(* Logix 5000 project; controller Generic 1768-L43 rev 16.2; software revision 15.01 *)

TASK T00_Main (continuous, watchdog 500 ms) : PZ_GenericMachine_AUTO, PZ_GenericMachine_MANUAL, P00_Control, P01_AXIS_00
TASK T02_AXIS_History (periodic, rate 48 ms, priority 10, watchdog 500 ms) : AXIS_EventLog

MODULES
   Local : 1768-L43 (1768Ctrl3Slot 0, Compact 0, rev 16.2)
      SERCOS : 1768-M04SE (1768 1, rev 16.1, MotionAsync RPI 25 ms, MotionEvent RPI 1000 ms, MotionSync RPI 2 ms)
END_MODULES

TYPE UDT_Axis_CMD :
STRUCT
   Enable : BOOL;   // 1=Turn Axis Servo Loop ON
   Disable : BOOL;   // 1=Turn Axis Servo Loop OFF
   Reset : BOOL;   // 1=Clear Axis Faults
   JogFWD : BOOL;   // 1=Jog Forward Direction
   JogREV : BOOL;   // 1=Jog Reverse Direction
   ReferenceREQ : BOOL;   // 1=Set Absolute Reference
END_STRUCT
END_TYPE

TYPE UDT_Axis_Data :
STRUCT
   MoveDir : DINT[8];
   MoveSpd : DINT[8];
   MoveAccel : DINT[8];
   MoveDecel : DINT[8];
   JogDir : DINT[8];
   JogSpd : DINT[8];
   JogAccel : DINT[8];
   JogDecel : DINT[8];
   Direction : DINT[8];
   Offset : REAL[4];
   Dwell : TIMER[16];
   JogTime : TIMER[16];
   InitSEQ : DINT;
   RunSEQ : DINT[4];
   StopSEQ : DINT;
   CamCalcSEQ : DINT;
END_STRUCT
END_TYPE

TYPE UDT_Axis_Status :
STRUCT
   Enabled : BOOL;   // 1=Axis Servo Loop is Active
   OK : BOOL;   // 1=Axis is NOT Faulted
   Auto : BOOL;   // 1=Axis has Attained the Auto Status Means
   Jogging : BOOL;   // 1=Axis is Jogging
   No_Motion : BOOL;   // 1=Axis is Stationary
   Homed : BOOL;   // 1=Axis has been Homed
   Axis_Selected : BOOL;   // 1=Axis to be Active When in Run Mode
   Gear_Active : BOOL;   // 1=Axis is Actively Geared to Another Axis
   Cam_Active : BOOL;   // 1=Axis is Actively Camming
   Move_Active : BOOL;   // 1=Axis is Actively Performing a Move
   Initialized : BOOL;   // 1=Axis has been Initialized
   ConfigComplete : BOOL;   // 1=Axis has been Configured
   ConfigState : DINT;   // Axis Configuration State
END_STRUCT
END_TYPE

TYPE UDT_AxisHistory_CTRL :
STRUCT
   Index : DINT;
   Date_Time : DINT[7];
   Next_Fault : DINT;
   MASR : MOTION_INSTRUCTION;
   Clear_History : BOOL;
   Latch_Bit : BOOL;
   ONS : DINT;
   SourceData : UDT_AxisHistory_DLM;
   Garbage : UDT_AxisHistory_DLM;
   FFL_FFU : CONTROL;
   Update_DLAY : TIMER;
   DLM_LoadDwell : TIMER[2];
END_STRUCT
END_TYPE

TYPE UDT_AxisHistory_DLM :
STRUCT
   SERCOS_NODE : DINT;
   Year : DINT;
   Month : DINT;
   Day : DINT;
   Hour : DINT;
   Minute : DINT;
   Second : DINT;
   GroupStatus : DINT;
   InhibStatus : DINT;
   GroupSynced : DINT;
   GroupFault : DINT;
   GroupOverlapFault : DINT;
   CSTLossFault : DINT;
   GroupTaskLoadingFault : DINT;
   GroupAxisFault : DINT;
   PhysicalAxisFault_Group : DINT;
   ModuleFault_Group : DINT;
   ConfigFault_Group : DINT;
   AxisFault : DINT;
   PhysicalAxisFault : DINT;
   ModuleFault : DINT;
   ConfigFault : DINT;
   ModuleFaults : DINT;
   ControlSyncFault : DINT;
   ModuleSyncFault : DINT;
   TimerEventFault : DINT;
   ModuleHardwareFault : DINT;
   SERCOSRingFault : DINT;
   AttributeErrorCode : DINT;
   AttributeErrorID : DINT;
   InhibitStatus : DINT;
   BusReadyStatus : DINT;
   DriveFault : DINT;
   PosSoftOvertravelFault : DINT;
   NegSoftOvertravelFault : DINT;
   PosHardOvertravelFault : DINT;
   NegHardOvertravelFault : DINT;
   MotFeedbackFault : DINT;
   MotFeedbackNoiseFault : DINT;
   AuxFeedbackFault : DINT;
   AuxFeedbackNoiseFault : DINT;
   DriveEnableInputFault : DINT;
   CommonBusFault : DINT;
   PreChargeOverloadFault : DINT;
   GroundShortFault : DINT;
   DriveHardFault : DINT;
   OverSpeedFault : DINT;
   OverloadFault : DINT;
   DriveOvertempFault : DINT;
   MotorOvertempFault : DINT;
   DriveCoolingFault : DINT;
   DriveControlVoltageFault : DINT;
   FeedbackFault : DINT;
   CommutationFault : DINT;
   DriveOvercurrentFault : DINT;
   DriveOvervoltageFault : DINT;
   DriveUndervoltageFault : DINT;
   PowerPhaseLossFault : DINT;
   PositionErrorFault : DINT;
   SERCOSFault : DINT;
   SERCOSErrorCode : DINT;
END_STRUCT
END_TYPE

TYPE UDT_Machine_COND :
STRUCT
   Networks_Ok : BOOL;
   ESTOP_OK : BOOL;
   GUARDS_OK : BOOL;
   LIGHT_CURTAIN_OK : BOOL;
   ALL_SAFETYs_OK : BOOL;
   All_Axes_Ok : BOOL;
   All_Axes_On : BOOL;
   All_Axes_Off : BOOL;
   All_Axes_Homed : BOOL;
   Home_Permissive : BOOL;
   Any_Line_Start_Pressed : BOOL;
   Any_Line_Stop_Pressed : BOOL;
   Any_Home_Request : BOOL;
   Any_Hold_Pressed : BOOL;
   Auto_Run_State_Active : BOOL;
   All_Axes_Running : BOOL;
   All_Axes_Initialized : BOOL;
   Init_Permissive : BOOL;
   All_Axes_Configured : BOOL;
   All_Axes_Bus_Ok : BOOL;
END_STRUCT
END_TYPE

TYPE UDT_Motion_Instructions :
STRUCT
   MASR : MOTION_INSTRUCTION;
   MAFR : MOTION_INSTRUCTION;
   MSO : MOTION_INSTRUCTION;
   MSF : MOTION_INSTRUCTION;
   MAH : MOTION_INSTRUCTION;
   MRP : MOTION_INSTRUCTION;
   MAJ : MOTION_INSTRUCTION[16];
   MAM : MOTION_INSTRUCTION[16];
   MAG : MOTION_INSTRUCTION[5];
   MCCP : MOTION_INSTRUCTION[5];
   MAPC : MOTION_INSTRUCTION[5];
   MAS : MOTION_INSTRUCTION[16];
   MCD : MOTION_INSTRUCTION;
   MAR : MOTION_INSTRUCTION;
   MDR : MOTION_INSTRUCTION;
END_STRUCT
END_TYPE

TYPE UDT_PhaseTimeout :
STRUCT
   Aborting : TIMER;
   Holding : TIMER;
   Resetting : TIMER;
   Restarting : TIMER;
   Running : TIMER;
   Stopping : TIMER;
END_STRUCT
END_TYPE

VAR_GLOBAL   (* controller tags *)
   AXIS_00 : AXIS_VIRTUAL;
   Axis_00_CMD : UDT_Axis_CMD := (Enable := 1);
   Axis_00_Data : UDT_Axis_Data := (MoveSpd[0] := 10, MoveSpd[1] := 20, MoveSpd[2] := 80, MoveSpd[3] := 90, MoveSpd[4] := 90, MoveAccel[0] := 50, MoveAccel[1] := 50, MoveAccel[2] := 30, MoveAccel[3] := 30, MoveAccel[4] := 40, MoveDecel[0] := 50, JogSpd[0] := 10, JogSpd[1] := 30, JogAccel[0] := 50, JogAccel[1] := 50, JogDecel[0] := 50, JogDecel[1] := 50, Direction[1] := 1, Direction[3] := 1, Dwell[0].PRE := 1500, Dwell[0].ACC := 1501, Dwell[0].EN := 1, Dwell[0].DN := 1, Dwell[1].PRE := 1500, Dwell[2].PRE := 1500, Dwell[2].ACC := 1502, Dwell[2].EN := 1, Dwell[2].DN := 1, Dwell[3].PRE := 1500, Dwell[3].ACC := 1501, Dwell[3].EN := 1, Dwell[3].DN := 1, Dwell[4].PRE := 1500, Dwell[4].ACC := 1500, Dwell[4].EN := 1, Dwell[4].DN := 1, JogTime[0].PRE := 5000, JogTime[1].PRE := 5000, JogTime[2].PRE := 5000, JogTime[3].PRE := 5000, JogTime[4].PRE := 5000);
   Axis_00_MI : UDT_Motion_Instructions := (MASR.FLAGS := 33554432, MAFR.FLAGS := 33554432, MSO.FLAGS := 536870912, MSO.DN := 1, MSO.STATE := 1, MSF.FLAGS := 536870912, MSF.DN := 1, MSF.STATUS := 2, MSF.STATE := 1, MAH.FLAGS := 33554432, MRP.FLAGS := 570425344, MRP.DN := 1, MAJ[0].FLAGS := 570425344, MAJ[0].DN := 1, MAJ[1].FLAGS := 33554432, MAJ[2].FLAGS := 33554432, MAJ[3].FLAGS := 570425344, MAJ[3].DN := 1, MAJ[4].FLAGS := 536870912, MAJ[4].DN := 1, MAM[0].FLAGS := 33554432, MAPC[0].FLAGS := 570425344, MAPC[0].DN := 1, MAS[0].FLAGS := 704643072, MAS[0].DN := 1, MAS[0].PC := 1, MAS[1].FLAGS := 33554432, MAS[2].FLAGS := 704643072, MAS[2].DN := 1, MAS[2].PC := 1, MAS[3].FLAGS := 704643072, MAS[3].DN := 1, MAS[3].PC := 1, MAS[4].FLAGS := 671088640, MAS[4].DN := 1, MAS[4].PC := 1);
   Axis_00_Status : UDT_Axis_Status := (Enabled := 1, OK := 1, Axis_Selected := 1, ConfigComplete := 1, ConfigState := 128);
   AXIS_01 : AXIS_SERVO_DRIVE;
   Axis_01_CMD : UDT_Axis_CMD;
   Axis_01_Data : UDT_Axis_Data := (MoveSpd[0] := 10, MoveSpd[1] := 20, MoveSpd[2] := 80, MoveSpd[3] := 90, MoveSpd[4] := 90, MoveAccel[0] := 50, MoveAccel[1] := 50, MoveAccel[2] := 30, MoveAccel[3] := 30, MoveAccel[4] := 40, MoveDecel[0] := 10, JogSpd[0] := 10, JogSpd[1] := 30, JogAccel[0] := 50, JogAccel[1] := 50, JogDecel[0] := 10, JogDecel[1] := 10, Direction[3] := 1, Dwell[0].PRE := 1500, Dwell[0].ACC := 1501, Dwell[0].EN := 1, Dwell[0].DN := 1, Dwell[1].PRE := 1500, Dwell[2].PRE := 1500, Dwell[2].ACC := 1502, Dwell[2].EN := 1, Dwell[2].DN := 1, Dwell[3].PRE := 1500, Dwell[3].ACC := 1501, Dwell[3].EN := 1, Dwell[3].DN := 1, Dwell[4].PRE := 1500, Dwell[4].ACC := 1500, Dwell[4].EN := 1, Dwell[4].DN := 1, JogTime[0].PRE := 5000, JogTime[1].PRE := 5000, JogTime[2].PRE := 5000, JogTime[3].PRE := 5000, JogTime[4].PRE := 5000);
   Axis_01_MI : UDT_Motion_Instructions := (MASR.FLAGS := 33554432, MAFR.FLAGS := 536870912, MAFR.DN := 1, MSO.FLAGS := 536870912, MSO.DN := 1, MSO.STATE := 1, MSF.FLAGS := 536870912, MSF.DN := 1, MSF.STATUS := 2, MSF.STATE := 1, MAH.FLAGS := 33554432, MAJ[0].FLAGS := 570425344, MAJ[0].DN := 1, MAJ[1].FLAGS := 33554432, MAJ[2].FLAGS := 33554432, MAJ[3].FLAGS := 570425344, MAJ[3].DN := 1, MAJ[4].FLAGS := 536870912, MAJ[4].DN := 1, MAM[0].FLAGS := 704643072, MAM[0].DN := 1, MAM[0].PC := 1, MAPC[0].FLAGS := 570425344, MAPC[0].DN := 1, MAS[0].FLAGS := 33554432, MAS[1].FLAGS := 33554432, MAS[2].FLAGS := 704643072, MAS[2].DN := 1, MAS[2].PC := 1, MAS[3].FLAGS := 704643072, MAS[3].DN := 1, MAS[3].PC := 1, MAS[4].FLAGS := 671088640, MAS[4].DN := 1, MAS[4].PC := 1);
   Axis_01_Status : UDT_Axis_Status := (OK := 1, Axis_Selected := 1, ConfigComplete := 1, ConfigState := 128);
   AXIS_02 : AXIS_SERVO_DRIVE;
   Axis_02_CMD : UDT_Axis_CMD;
   Axis_02_Data : UDT_Axis_Data := (MoveSpd[0] := 10, MoveSpd[1] := 20, MoveSpd[2] := 80, MoveSpd[3] := 90, MoveSpd[4] := 90, MoveAccel[0] := 50, MoveAccel[1] := 50, MoveAccel[2] := 30, MoveAccel[3] := 30, MoveAccel[4] := 40, MoveDecel[0] := 10, JogSpd[0] := 10, JogSpd[1] := 30, JogAccel[0] := 50, JogAccel[1] := 50, JogDecel[0] := 10, JogDecel[1] := 10, Direction[3] := 1, Dwell[0].PRE := 1500, Dwell[1].PRE := 1500, Dwell[2].PRE := 1500, Dwell[2].ACC := 1501, Dwell[2].EN := 1, Dwell[2].DN := 1, Dwell[3].PRE := 1500, Dwell[3].ACC := 1501, Dwell[3].EN := 1, Dwell[3].DN := 1, Dwell[4].PRE := 1500, Dwell[4].ACC := 1502, Dwell[4].EN := 1, Dwell[4].DN := 1, JogTime[0].PRE := 5000, JogTime[0].ACC := 4648, JogTime[0].EN := 1, JogTime[0].TT := 1, JogTime[1].PRE := 5000, JogTime[2].PRE := 5000, JogTime[3].PRE := 5000, JogTime[4].PRE := 5000);
   Axis_02_MI : UDT_Motion_Instructions := (MASR.FLAGS := 33554432, MAFR.FLAGS := 536870912, MAFR.DN := 1, MSO.FLAGS := 536870912, MSO.DN := 1, MSO.STATE := 1, MSF.FLAGS := 536870912, MSF.DN := 1, MSF.STATUS := 2, MSF.STATE := 1, MAH.FLAGS := 33554432, MAJ[0].FLAGS := 570425344, MAJ[0].DN := 1, MAJ[1].FLAGS := 33554432, MAJ[2].FLAGS := 33554432, MAJ[3].FLAGS := 570425344, MAJ[3].DN := 1, MAJ[4].FLAGS := 536870912, MAJ[4].DN := 1, MAM[0].FLAGS := 704643072, MAM[0].DN := 1, MAM[0].PC := 1, MAS[0].FLAGS := 33554432, MAS[1].FLAGS := 33554432, MAS[2].FLAGS := 704643072, MAS[2].DN := 1, MAS[2].PC := 1, MAS[3].FLAGS := 704643072, MAS[3].DN := 1, MAS[3].PC := 1, MAS[4].FLAGS := 671088640, MAS[4].DN := 1, MAS[4].PC := 1);
   Axis_02_Status : UDT_Axis_Status := (Axis_Selected := 1, ConfigComplete := 1, ConfigState := 128);
   AXIS_03 : AXIS_SERVO_DRIVE;
   Axis_03_CMD : UDT_Axis_CMD;
   Axis_03_Data : UDT_Axis_Data := (MoveSpd[0] := 10, MoveSpd[1] := 20, MoveSpd[2] := 80, MoveSpd[3] := 90, MoveSpd[4] := 90, MoveAccel[0] := 50, MoveAccel[1] := 50, MoveAccel[2] := 30, MoveAccel[3] := 30, MoveAccel[4] := 40, MoveDecel[0] := 10, JogSpd[0] := 10, JogSpd[1] := 30, JogAccel[0] := 50, JogAccel[1] := 50, JogDecel[0] := 10, JogDecel[1] := 10, Direction[3] := 1, Dwell[0].PRE := 1500, Dwell[1].PRE := 1500, Dwell[2].PRE := 1500, Dwell[2].ACC := 1501, Dwell[2].EN := 1, Dwell[2].DN := 1, Dwell[3].PRE := 1500, Dwell[3].ACC := 1501, Dwell[3].EN := 1, Dwell[3].DN := 1, Dwell[4].PRE := 1500, Dwell[4].ACC := 1502, Dwell[4].EN := 1, Dwell[4].DN := 1, JogTime[0].PRE := 5000, JogTime[0].ACC := 4648, JogTime[0].EN := 1, JogTime[0].TT := 1, JogTime[1].PRE := 5000, JogTime[2].PRE := 5000, JogTime[3].PRE := 5000, JogTime[4].PRE := 5000);
   Axis_03_MI : UDT_Motion_Instructions := (MASR.FLAGS := 33554432, MAFR.FLAGS := 536870912, MAFR.DN := 1, MSO.FLAGS := 536870912, MSO.DN := 1, MSO.STATE := 1, MSF.FLAGS := 536870912, MSF.DN := 1, MSF.STATUS := 2, MSF.STATE := 1, MAH.FLAGS := 33554432, MAJ[0].FLAGS := 570425344, MAJ[0].DN := 1, MAJ[1].FLAGS := 33554432, MAJ[2].FLAGS := 33554432, MAJ[3].FLAGS := 570425344, MAJ[3].DN := 1, MAJ[4].FLAGS := 536870912, MAJ[4].DN := 1, MAM[0].FLAGS := 704643072, MAM[0].DN := 1, MAM[0].PC := 1, MAS[0].FLAGS := 33554432, MAS[1].FLAGS := 33554432, MAS[2].FLAGS := 704643072, MAS[2].DN := 1, MAS[2].PC := 1, MAS[3].FLAGS := 704643072, MAS[3].DN := 1, MAS[3].PC := 1, MAS[4].FLAGS := 671088640, MAS[4].DN := 1, MAS[4].PC := 1);
   Axis_03_Status : UDT_Axis_Status := (Axis_Selected := 1, ConfigComplete := 1, ConfigState := 128);
   AXIS_04 : AXIS_SERVO_DRIVE;
   Axis_04_CMD : UDT_Axis_CMD;
   Axis_04_Data : UDT_Axis_Data := (MoveSpd[0] := 10, MoveSpd[1] := 20, MoveSpd[2] := 80, MoveSpd[3] := 90, MoveSpd[4] := 90, MoveAccel[0] := 50, MoveAccel[1] := 50, MoveAccel[2] := 30, MoveAccel[3] := 30, MoveAccel[4] := 40, MoveDecel[0] := 10, JogSpd[0] := 10, JogSpd[1] := 30, JogAccel[0] := 50, JogAccel[1] := 50, JogDecel[0] := 10, JogDecel[1] := 10, Direction[3] := 1, Dwell[0].PRE := 1500, Dwell[1].PRE := 1500, Dwell[2].PRE := 1500, Dwell[2].ACC := 1501, Dwell[2].EN := 1, Dwell[2].DN := 1, Dwell[3].PRE := 1500, Dwell[3].ACC := 1501, Dwell[3].EN := 1, Dwell[3].DN := 1, Dwell[4].PRE := 1500, Dwell[4].ACC := 1502, Dwell[4].EN := 1, Dwell[4].DN := 1, JogTime[0].PRE := 5000, JogTime[0].ACC := 4648, JogTime[0].EN := 1, JogTime[0].TT := 1, JogTime[1].PRE := 5000, JogTime[2].PRE := 5000, JogTime[3].PRE := 5000, JogTime[4].PRE := 5000);
   Axis_04_MI : UDT_Motion_Instructions := (MASR.FLAGS := 33554432, MAFR.FLAGS := 536870912, MAFR.DN := 1, MSO.FLAGS := 536870912, MSO.DN := 1, MSO.STATE := 1, MSF.FLAGS := 536870912, MSF.DN := 1, MSF.STATUS := 2, MSF.STATE := 1, MAH.FLAGS := 33554432, MAJ[0].FLAGS := 570425344, MAJ[0].DN := 1, MAJ[1].FLAGS := 33554432, MAJ[2].FLAGS := 33554432, MAJ[3].FLAGS := 570425344, MAJ[3].DN := 1, MAJ[4].FLAGS := 536870912, MAJ[4].DN := 1, MAM[0].FLAGS := 704643072, MAM[0].DN := 1, MAM[0].PC := 1, MAS[0].FLAGS := 33554432, MAS[1].FLAGS := 33554432, MAS[2].FLAGS := 704643072, MAS[2].DN := 1, MAS[2].PC := 1, MAS[3].FLAGS := 704643072, MAS[3].DN := 1, MAS[3].PC := 1, MAS[4].FLAGS := 671088640, MAS[4].DN := 1, MAS[4].PC := 1);
   Axis_04_Status : UDT_Axis_Status := (Axis_Selected := 1, ConfigComplete := 1, ConfigState := 128);
   AXIS_Servo_Generic : AXIS_SERVO_DRIVE;
   C_pi : REAL := 3.1415927;
   ClearFaultDelay : TIMER := (PRE := 250);
   GenericMachine_COND : UDT_Machine_COND := (Networks_Ok := 1, ESTOP_OK := 1, GUARDS_OK := 1, LIGHT_CURTAIN_OK := 1, ALL_SAFETYs_OK := 1, All_Axes_Off := 1, Init_Permissive := 1, All_Axes_Configured := 1, All_Axes_Bus_Ok := 1);
   GUI_Axis_01_JogFwdREQ : BOOL;
   GUI_Axis_01_JogRevREQ : BOOL;
   GUI_Axis_01_ReferenceREQ : BOOL;
   GUI_Axis_02_JogFwdREQ : BOOL;
   GUI_Axis_02_JogRevREQ : BOOL;
   GUI_Axis_02_ReferenceREQ : BOOL;
   GUI_Axis_03_JogFwdREQ : BOOL;
   GUI_Axis_03_JogRevREQ : BOOL;
   GUI_Axis_03_ReferenceREQ : BOOL;
   GUI_Axis_04_JogFwdREQ : BOOL;
   GUI_Axis_04_JogRevREQ : BOOL;
   GUI_Axis_04_ReferenceREQ : BOOL;
   GUI_HoldRequest : BOOL;
   GUI_JogFwdRequest : BOOL;
   GUI_JogRevRequest : BOOL;
   GUI_ManualABSrefStatDISP : DINT := 1;
   GUI_ManualAxisSelect : DINT;
   GUI_ManualControlRequest : BOOL;
   GUI_ManualPositionDISP : REAL := 0.334165;
   GUI_ManualSASDISP : DINT;
   GUI_ManualVelocityDISP : REAL;
   GUI_ReferenceREQ : BOOL;
   GUI_RunSPD_NI : DINT := 5;
   GUI_ServoReReferenceRequest : BOOL;
   GUI_StartRequest : BOOL;
   GUI_StopRequest : BOOL;
   ManualControl : BOOL;
   MASK : DINT := -1;
   MotionGroup : MOTION_GROUP;
   PhaseTimout : UDT_PhaseTimeout := (Aborting.PRE := 5000, Holding.PRE := 5000, Resetting.PRE := 5000, Restarting.PRE := 5000, Stopping.PRE := 5000);
   PowerUP_TMR : TIMER := (PRE := 10000, ACC := 10000);
   PZ_GenericMachine_AUTO : PHASE := (State := 1024, Aborted := 1);
   PZ_GenericMachine_MANUAL : PHASE := (State := 512, Stopped := 1);
END_VAR

PROGRAM AXIS_EventLog   (* main routine R00_Dispatch *)
VAR
   EL_CTRL_1 : UDT_AxisHistory_CTRL := (Date_Time[0] := 1998, Date_Time[1] := 1, Date_Time[2] := 4, Date_Time[3] := 14, Date_Time[4] := 48, Date_Time[5] := 48, Date_Time[6] := 956843, SourceData.SERCOS_NODE := 1, SourceData.Year := 1998, SourceData.Month := 1, SourceData.Day := 4, SourceData.Hour := 14, SourceData.Minute := 48, SourceData.Second := 48, SourceData.GroupStatus := 16#0000_0006, SourceData.GroupSynced := 1, SourceData.GroupAxisFault := 16#0000_0001, SourceData.PhysicalAxisFault_Group := 1, SourceData.AxisFault := 16#0000_0001, SourceData.PhysicalAxisFault := 1, SourceData.DriveFault := 16#0800_0000, SourceData.PositionErrorFault := 1, FFL_FFU.LEN := 51, FFL_FFU.POS := 50, Update_DLAY.PRE := 24, DLM_LoadDwell[0].PRE := 1000, DLM_LoadDwell[1].PRE := 1000);
   EL_CTRL_2 : UDT_AxisHistory_CTRL := (Date_Time[0] := 1998, Date_Time[1] := 1, Date_Time[2] := 4, Date_Time[3] := 14, Date_Time[4] := 54, Date_Time[5] := 19, Date_Time[6] := 52840, Next_Fault := 3, ONS := 1, SourceData.SERCOS_NODE := 2, SourceData.Year := 1998, SourceData.Month := 1, SourceData.Day := 4, SourceData.Hour := 14, SourceData.Minute := 54, SourceData.Second := 19, SourceData.GroupStatus := 16#0000_0006, SourceData.GroupSynced := 1, SourceData.GroupAxisFault := 16#0000_0001, SourceData.PhysicalAxisFault_Group := 1, SourceData.AxisFault := 16#0000_0001, SourceData.PhysicalAxisFault := 1, SourceData.DriveFault := 16#0800_0000, SourceData.PositionErrorFault := 1, FFL_FFU.LEN := 51, FFL_FFU.POS := 50, Update_DLAY.PRE := 24, Update_DLAY.ACC := 48, Update_DLAY.EN := 1, Update_DLAY.DN := 1, DLM_LoadDwell[0].PRE := 1000, DLM_LoadDwell[1].PRE := 1000);
   EL_CTRL_3 : UDT_AxisHistory_CTRL := (Date_Time[0] := 1998, Date_Time[1] := 1, Date_Time[2] := 1, Date_Time[3] := 15, Date_Time[4] := 41, Date_Time[5] := 17, Date_Time[6] := 485526, FFL_FFU.LEN := 51, FFL_FFU.POS := 50, FFL_FFU.EN := 1, FFL_FFU.EU := 1, Update_DLAY.PRE := 24, DLM_LoadDwell[0].PRE := 1000, DLM_LoadDwell[1].PRE := 1000);
   EL_CTRL_4 : UDT_AxisHistory_CTRL := (Date_Time[0] := 1998, Date_Time[1] := 1, Date_Time[2] := 1, Date_Time[3] := 15, Date_Time[4] := 41, Date_Time[5] := 17, Date_Time[6] := 437605, FFL_FFU.LEN := 51, FFL_FFU.POS := 50, FFL_FFU.EN := 1, FFL_FFU.EU := 1, Update_DLAY.PRE := 24, DLM_LoadDwell[0].PRE := 1000, DLM_LoadDwell[1].PRE := 1000);
   EL_CTRL_5 : UDT_AxisHistory_CTRL := (Date_Time[0] := 1998, Date_Time[1] := 1, Date_Time[2] := 1, Date_Time[3] := 15, Date_Time[4] := 41, Date_Time[5] := 17, Date_Time[6] := 438340, FFL_FFU.LEN := 51, FFL_FFU.POS := 50, FFL_FFU.EN := 1, FFL_FFU.EU := 1, Update_DLAY.PRE := 24, DLM_LoadDwell[0].PRE := 1000, DLM_LoadDwell[1].PRE := 1000);
   EL_CTRL_6 : UDT_AxisHistory_CTRL := (FFL_FFU.LEN := 51, FFL_FFU.POS := 50, FFL_FFU.EN := 1, FFL_FFU.EU := 1, Update_DLAY.PRE := 24, DLM_LoadDwell[0].PRE := 1000, DLM_LoadDwell[1].PRE := 1000);
   EL_CTRL_7 : UDT_AxisHistory_CTRL := (Date_Time[0] := 2006, Date_Time[1] := 2, Date_Time[2] := 9, Date_Time[3] := 17, Date_Time[4] := 41, Date_Time[5] := 26, Date_Time[6] := 391260, SourceData.SERCOS_NODE := 7, SourceData.Year := 2006, SourceData.Month := 2, SourceData.Day := 9, SourceData.Hour := 17, SourceData.Minute := 41, SourceData.Second := 26, SourceData.GroupStatus := 16#0000_0006, SourceData.GroupSynced := 1, SourceData.GroupAxisFault := 16#0000_0001, SourceData.PhysicalAxisFault_Group := 1, SourceData.AxisFault := 16#0000_0001, SourceData.PhysicalAxisFault := 1, SourceData.DriveFault := 16#0800_0000, SourceData.PositionErrorFault := 1, FFL_FFU.LEN := 51, FFL_FFU.POS := 50, FFL_FFU.EN := 1, FFL_FFU.EU := 1, Update_DLAY.PRE := 24, DLM_LoadDwell[0].PRE := 1000, DLM_LoadDwell[1].PRE := 1000);
   EL_CTRL_8 : UDT_AxisHistory_CTRL := (Date_Time[0] := 2006, Date_Time[1] := 2, Date_Time[2] := 9, Date_Time[3] := 17, Date_Time[4] := 43, Date_Time[5] := 28, Date_Time[6] := 567606, SourceData.SERCOS_NODE := 8, SourceData.Year := 2006, SourceData.Month := 2, SourceData.Day := 9, SourceData.Hour := 17, SourceData.Minute := 43, SourceData.Second := 28, SourceData.GroupStatus := 16#0000_0006, SourceData.GroupSynced := 1, SourceData.GroupAxisFault := 16#0000_0001, SourceData.PhysicalAxisFault_Group := 1, SourceData.AxisFault := 16#0000_0001, SourceData.PhysicalAxisFault := 1, SourceData.DriveFault := 16#0800_0000, SourceData.PositionErrorFault := 1, FFL_FFU.LEN := 51, FFL_FFU.POS := 50, FFL_FFU.EN := 1, FFL_FFU.EU := 1, Update_DLAY.PRE := 24, DLM_LoadDwell[0].PRE := 1000, DLM_LoadDwell[1].PRE := 1000);
   EL_SaveSEQ : DINT;
   EventINDEX : DINT;
   EventLog_N1 : UDT_AxisHistory_DLM[51];
   EventLog_N2 : UDT_AxisHistory_DLM[51];
   EventLog_N3 : UDT_AxisHistory_DLM[51];
   EventLog_N4 : UDT_AxisHistory_DLM[51];
   EventLog_N5 : UDT_AxisHistory_DLM[51];
   EventLog_N6 : UDT_AxisHistory_DLM[51];
   EventLog_N7 : UDT_AxisHistory_DLM[51];
   EventLog_N8 : UDT_AxisHistory_DLM[51];
   GUI_DataDisplay : UDT_AxisHistory_DLM;
   GUI_DataLogModel : UDT_AxisHistory_DLM := (SERCOS_NODE := -1, Year := -1, Month := -1, Day := -1, Hour := -1, Minute := -1, Second := -1, GroupStatus := 16#ffff_ffff, InhibStatus := -1, GroupSynced := -1, GroupFault := 16#ffff_ffff, GroupOverlapFault := -1, CSTLossFault := -1, GroupTaskLoadingFault := -1, GroupAxisFault := 16#ffff_ffff, PhysicalAxisFault_Group := -1, ModuleFault_Group := -1, ConfigFault_Group := -1, AxisFault := 16#ffff_ffff, PhysicalAxisFault := -1, ModuleFault := -1, ConfigFault := -1, ModuleFaults := 16#ffff_ffff, ControlSyncFault := -1, ModuleSyncFault := -1, TimerEventFault := -1, ModuleHardwareFault := -1, SERCOSRingFault := -1, AttributeErrorCode := 16#ffff_ffff, AttributeErrorID := 16#ffff_ffff, InhibitStatus := -1, BusReadyStatus := -1, DriveFault := 16#ffff_ffff, PosSoftOvertravelFault := -1, NegSoftOvertravelFault := -1, PosHardOvertravelFault := -1, NegHardOvertravelFault := -1, MotFeedbackFault := -1, MotFeedbackNoiseFault := -1, AuxFeedbackFault := -1, AuxFeedbackNoiseFault := -1, DriveEnableInputFault := -1, CommonBusFault := -1, PreChargeOverloadFault := -1, GroundShortFault := -1, DriveHardFault := -1, OverSpeedFault := -1, OverloadFault := -1, DriveOvertempFault := -1, MotorOvertempFault := -1, DriveCoolingFault := -1, DriveControlVoltageFault := -1, FeedbackFault := -1, CommutationFault := -1, DriveOvercurrentFault := -1, DriveOvervoltageFault := -1, DriveUndervoltageFault := -1, PowerPhaseLossFault := -1, PositionErrorFault := -1, SERCOSFault := -1,
        SERCOSErrorCode := 16#ffff_ffff);
   GUI_EventLogSaving : BOOL;
   GUI_IndexSelect : DINT := 48;
   GUI_NodeSelect : DINT := 8;
   GUI_SaveEventLog : BOOL;
   LogLength : DINT := 51;
   Motion_Group : ALIAS FOR MotionGroup;
   PowerUP_TMR : TIMER := (PRE := 10000, ACC := 10032);
   Servo_Axis_Node_1 : ALIAS FOR AXIS_01;
   Servo_Axis_Node_2 : ALIAS FOR AXIS_02;
   Servo_Axis_Node_3 : ALIAS FOR AXIS_03;
   Servo_Axis_Node_4 : ALIAS FOR AXIS_04;
   Servo_Axis_Node_5 : ALIAS FOR AXIS_Servo_Generic;
   Servo_Axis_Node_6 : ALIAS FOR AXIS_Servo_Generic;
   Servo_Axis_Node_7 : ALIAS FOR AXIS_Servo_Generic;
   Servo_Axis_Node_8 : ALIAS FOR AXIS_Servo_Generic;
END_VAR

ROUTINE R00_Dispatch   (* ladder *)
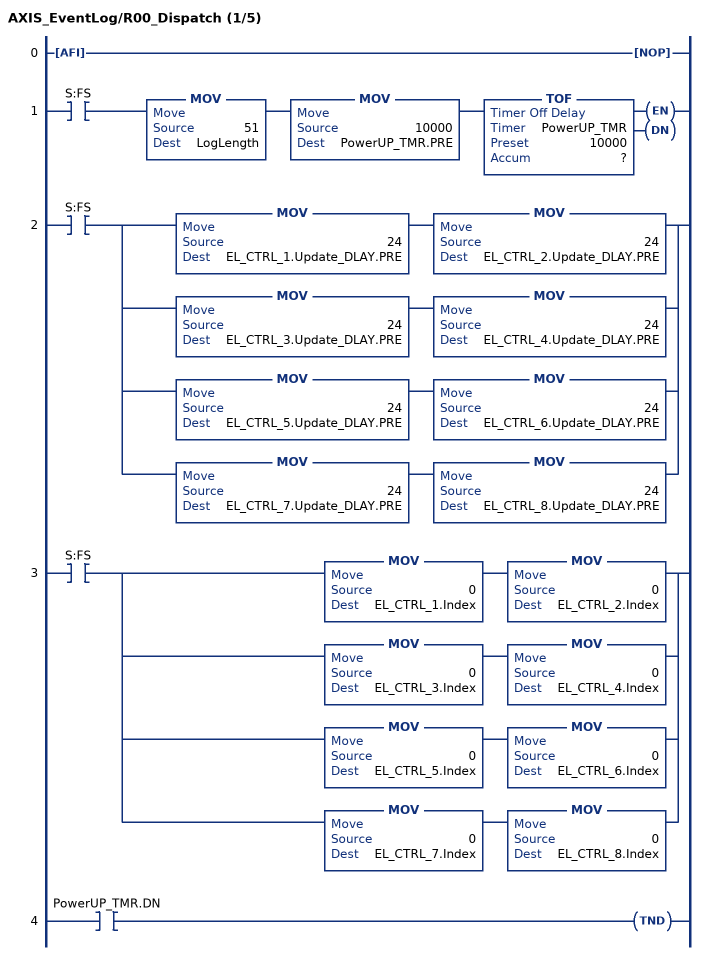
   0: AFI()NOP();
   1: XIC(S:FS)MOV(51,LogLength)MOV(10000,PowerUP_TMR.PRE)TOF(PowerUP_TMR,?,?);
   2: XIC(S:FS)[MOV(24,EL_CTRL_1.Update_DLAY.PRE) MOV(24,EL_CTRL_2.Update_DLAY.PRE) ,MOV(24,EL_CTRL_3.Update_DLAY.PRE) MOV(24,EL_CTRL_4.Update_DLAY.PRE) ,MOV(24,EL_CTRL_5.Update_DLAY.PRE) MOV(24,EL_CTRL_6.Update_DLAY.PRE) ,MOV(24,EL_CTRL_7.Update_DLAY.PRE) MOV(24,EL_CTRL_8.Update_DLAY.PRE) ];
   3: XIC(S:FS)[MOV(0,EL_CTRL_1.Index) MOV(0,EL_CTRL_2.Index) ,MOV(0,EL_CTRL_3.Index) MOV(0,EL_CTRL_4.Index) ,MOV(0,EL_CTRL_5.Index) MOV(0,EL_CTRL_6.Index) ,MOV(0,EL_CTRL_7.Index) MOV(0,EL_CTRL_8.Index) ];
   4: XIC(PowerUP_TMR.DN)TND();
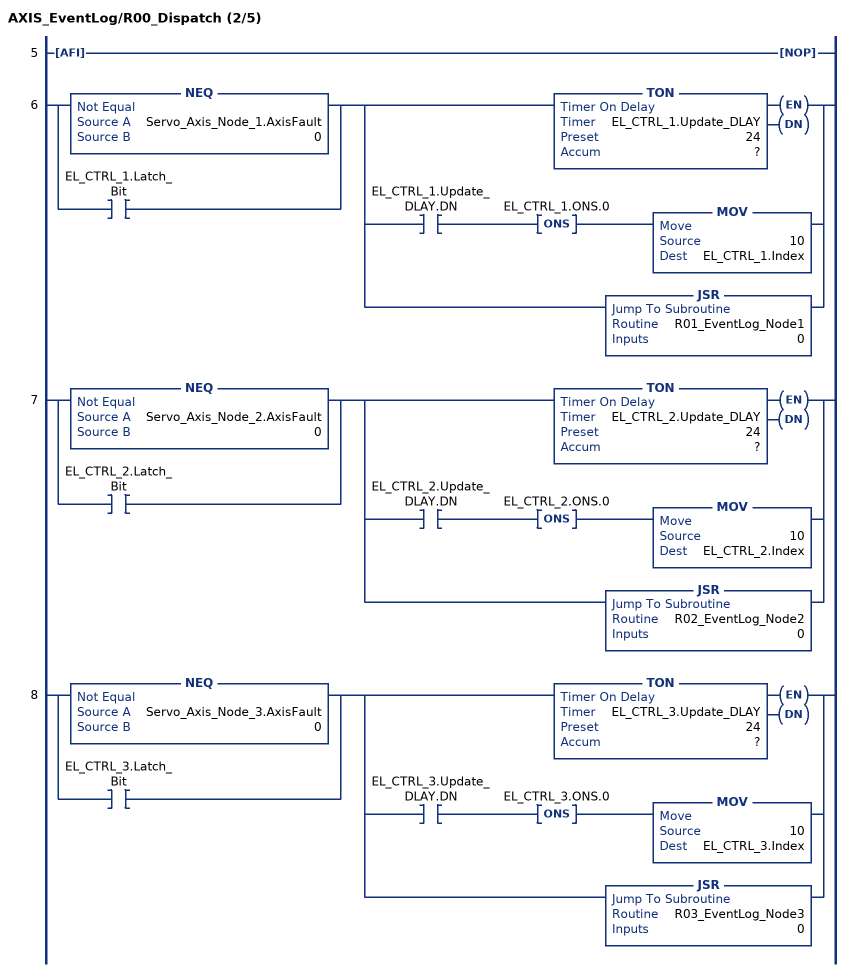
   5: AFI()NOP();
   6: [NEQ(Servo_Axis_Node_1.AxisFault,0) ,XIC(EL_CTRL_1.Latch_Bit) ][TON(EL_CTRL_1.Update_DLAY,?,?) ,XIC(EL_CTRL_1.Update_DLAY.DN) ONS(EL_CTRL_1.ONS.0) MOV(10,EL_CTRL_1.Index) ,JSR(R01_EventLog_Node1,0) ];
   7: [NEQ(Servo_Axis_Node_2.AxisFault,0) ,XIC(EL_CTRL_2.Latch_Bit) ][TON(EL_CTRL_2.Update_DLAY,?,?) ,XIC(EL_CTRL_2.Update_DLAY.DN) ONS(EL_CTRL_2.ONS.0) MOV(10,EL_CTRL_2.Index) ,JSR(R02_EventLog_Node2,0) ];
   8: [NEQ(Servo_Axis_Node_3.AxisFault,0) ,XIC(EL_CTRL_3.Latch_Bit) ][TON(EL_CTRL_3.Update_DLAY,?,?) ,XIC(EL_CTRL_3.Update_DLAY.DN) ONS(EL_CTRL_3.ONS.0) MOV(10,EL_CTRL_3.Index) ,JSR(R03_EventLog_Node3,0) ];
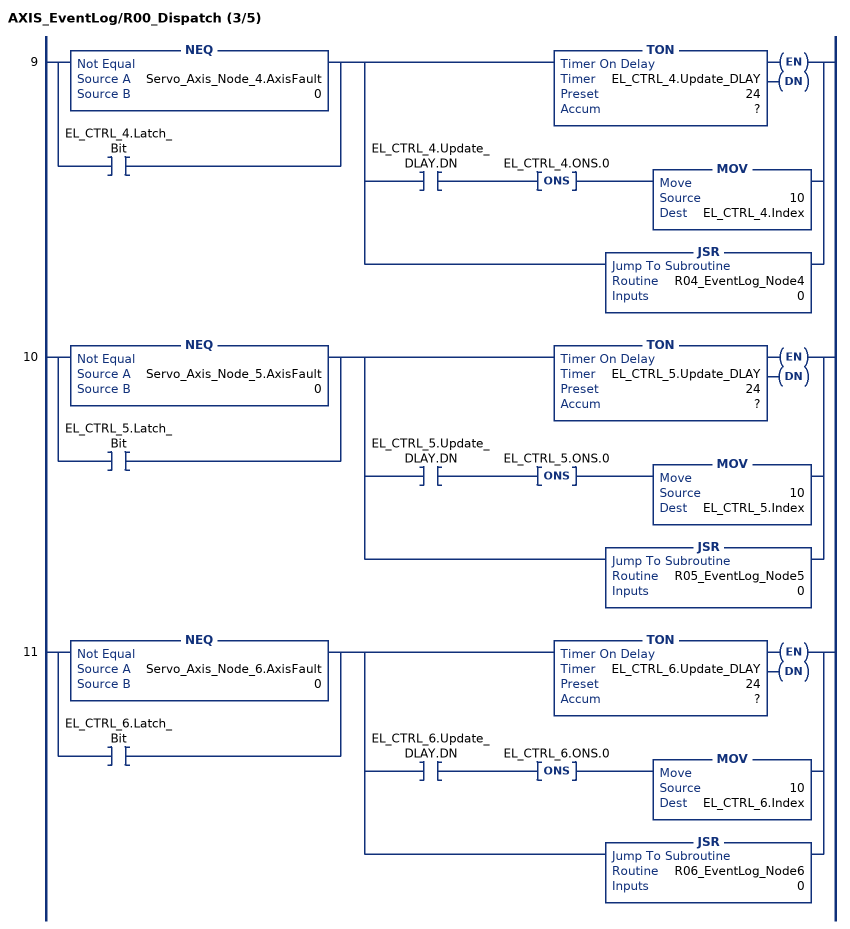
   9: [NEQ(Servo_Axis_Node_4.AxisFault,0) ,XIC(EL_CTRL_4.Latch_Bit) ][TON(EL_CTRL_4.Update_DLAY,?,?) ,XIC(EL_CTRL_4.Update_DLAY.DN) ONS(EL_CTRL_4.ONS.0) MOV(10,EL_CTRL_4.Index) ,JSR(R04_EventLog_Node4,0) ];
   10: [NEQ(Servo_Axis_Node_5.AxisFault,0) ,XIC(EL_CTRL_5.Latch_Bit) ][TON(EL_CTRL_5.Update_DLAY,?,?) ,XIC(EL_CTRL_5.Update_DLAY.DN) ONS(EL_CTRL_5.ONS.0) MOV(10,EL_CTRL_5.Index) ,JSR(R05_EventLog_Node5,0) ];
   11: [NEQ(Servo_Axis_Node_6.AxisFault,0) ,XIC(EL_CTRL_6.Latch_Bit) ][TON(EL_CTRL_6.Update_DLAY,?,?) ,XIC(EL_CTRL_6.Update_DLAY.DN) ONS(EL_CTRL_6.ONS.0) MOV(10,EL_CTRL_6.Index) ,JSR(R06_EventLog_Node6,0) ];
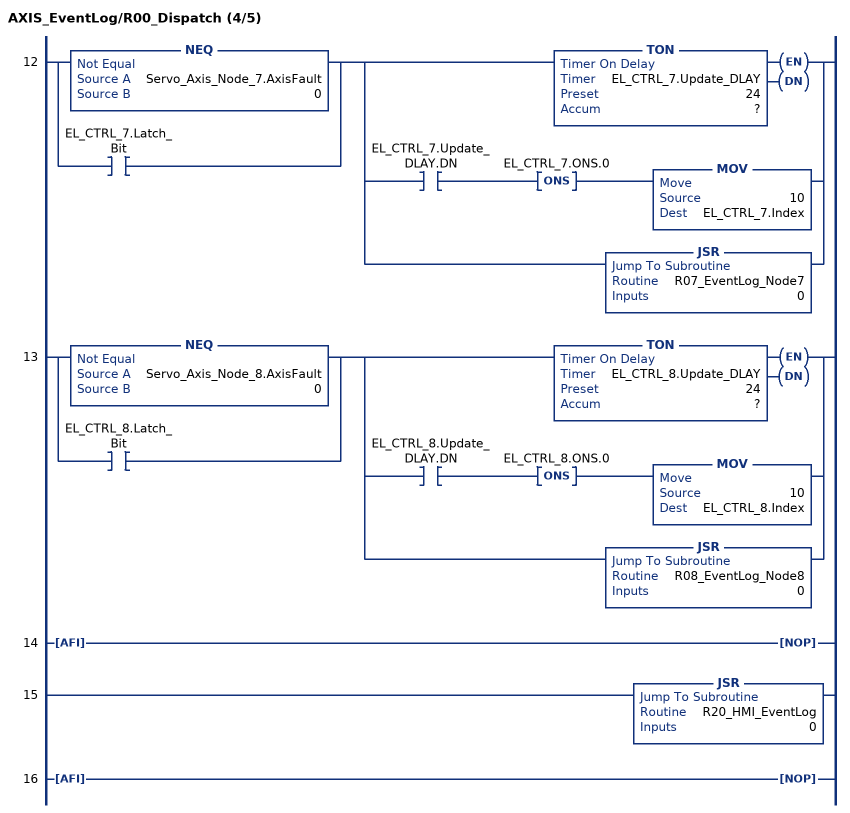
   12: [NEQ(Servo_Axis_Node_7.AxisFault,0) ,XIC(EL_CTRL_7.Latch_Bit) ][TON(EL_CTRL_7.Update_DLAY,?,?) ,XIC(EL_CTRL_7.Update_DLAY.DN) ONS(EL_CTRL_7.ONS.0) MOV(10,EL_CTRL_7.Index) ,JSR(R07_EventLog_Node7,0) ];
   13: [NEQ(Servo_Axis_Node_8.AxisFault,0) ,XIC(EL_CTRL_8.Latch_Bit) ][TON(EL_CTRL_8.Update_DLAY,?,?) ,XIC(EL_CTRL_8.Update_DLAY.DN) ONS(EL_CTRL_8.ONS.0) MOV(10,EL_CTRL_8.Index) ,JSR(R08_EventLog_Node8,0) ];
   14: AFI()NOP();
   15: JSR(R20_HMI_EventLog,0);
   16: AFI()NOP();
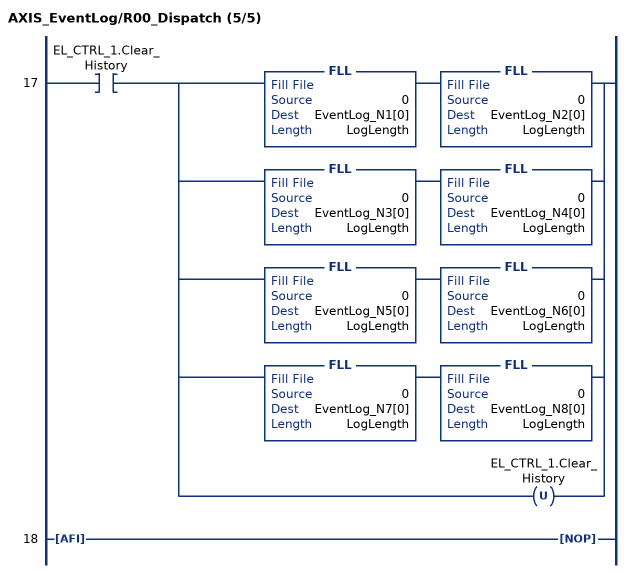
   17: XIC(EL_CTRL_1.Clear_History)[FLL(0,EventLog_N1[0],LogLength) FLL(0,EventLog_N2[0],LogLength) ,FLL(0,EventLog_N3[0],LogLength) FLL(0,EventLog_N4[0],LogLength) ,FLL(0,EventLog_N5[0],LogLength) FLL(0,EventLog_N6[0],LogLength) ,FLL(0,EventLog_N7[0],LogLength) FLL(0,EventLog_N8[0],LogLength) ,OTU(EL_CTRL_1.Clear_History) ];
   18: AFI()NOP();
END_ROUTINE

ROUTINE R01_EventLog_Node1   (* ladder *)
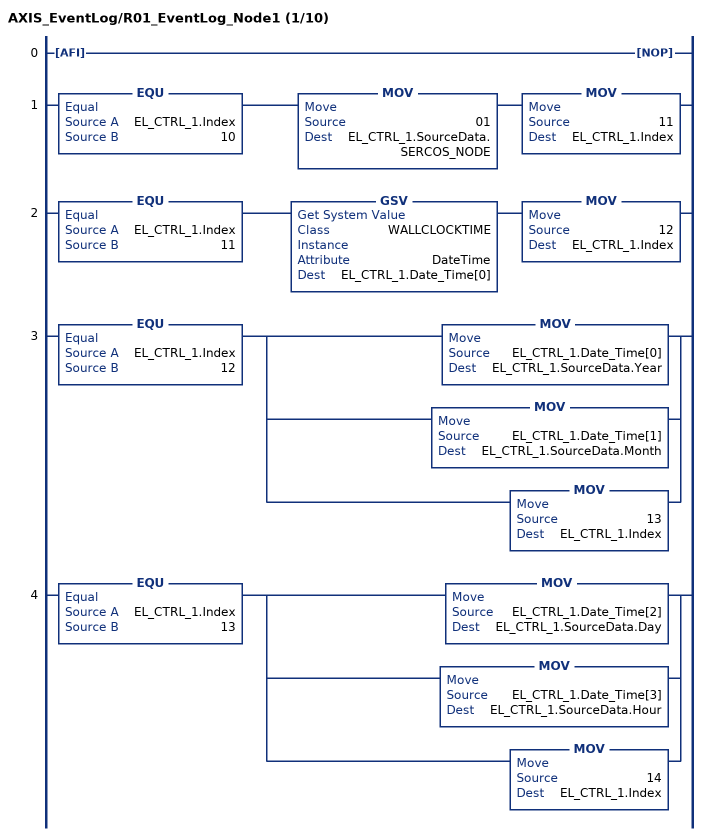
   0: AFI()NOP();
   1: EQU(EL_CTRL_1.Index,10)MOV(01,EL_CTRL_1.SourceData.SERCOS_NODE)MOV(11,EL_CTRL_1.Index);
   2: EQU(EL_CTRL_1.Index,11)GSV(WALLCLOCKTIME,,DateTime,EL_CTRL_1.Date_Time[0])MOV(12,EL_CTRL_1.Index);
   3: EQU(EL_CTRL_1.Index,12)[MOV(EL_CTRL_1.Date_Time[0],EL_CTRL_1.SourceData.Year) ,MOV(EL_CTRL_1.Date_Time[1],EL_CTRL_1.SourceData.Month) ,MOV(13,EL_CTRL_1.Index) ];
   4: EQU(EL_CTRL_1.Index,13)[MOV(EL_CTRL_1.Date_Time[2],EL_CTRL_1.SourceData.Day) ,MOV(EL_CTRL_1.Date_Time[3],EL_CTRL_1.SourceData.Hour) ,MOV(14,EL_CTRL_1.Index) ];
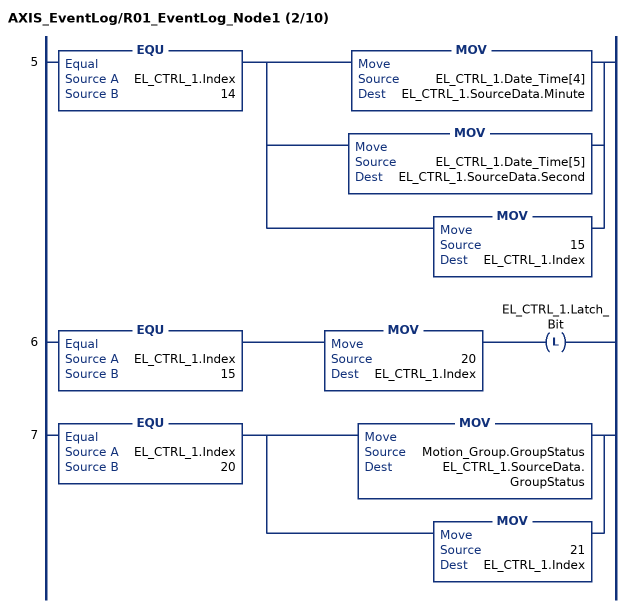
   5: EQU(EL_CTRL_1.Index,14)[MOV(EL_CTRL_1.Date_Time[4],EL_CTRL_1.SourceData.Minute) ,MOV(EL_CTRL_1.Date_Time[5],EL_CTRL_1.SourceData.Second) ,MOV(15,EL_CTRL_1.Index) ];
   6: EQU(EL_CTRL_1.Index,15)MOV(20,EL_CTRL_1.Index)OTL(EL_CTRL_1.Latch_Bit);
   7: EQU(EL_CTRL_1.Index,20)[MOV(Motion_Group.GroupStatus,EL_CTRL_1.SourceData.GroupStatus) ,MOV(21,EL_CTRL_1.Index) ];
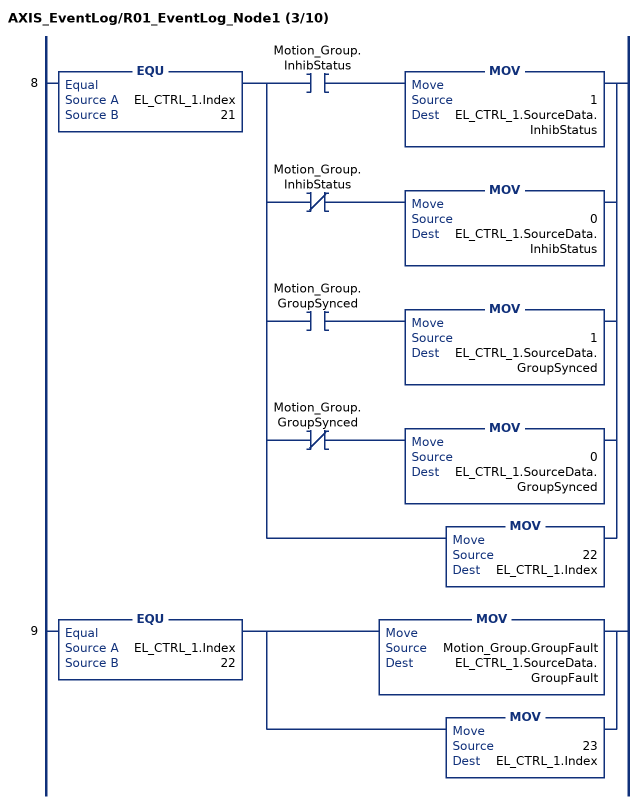
   8: EQU(EL_CTRL_1.Index,21)[XIC(Motion_Group.InhibStatus) MOV(1,EL_CTRL_1.SourceData.InhibStatus) ,XIO(Motion_Group.InhibStatus) MOV(0,EL_CTRL_1.SourceData.InhibStatus) ,XIC(Motion_Group.GroupSynced) MOV(1,EL_CTRL_1.SourceData.GroupSynced) ,XIO(Motion_Group.GroupSynced) MOV(0,EL_CTRL_1.SourceData.GroupSynced) ,MOV(22,EL_CTRL_1.Index) ];
   9: EQU(EL_CTRL_1.Index,22)[MOV(Motion_Group.GroupFault,EL_CTRL_1.SourceData.GroupFault) ,MOV(23,EL_CTRL_1.Index) ];
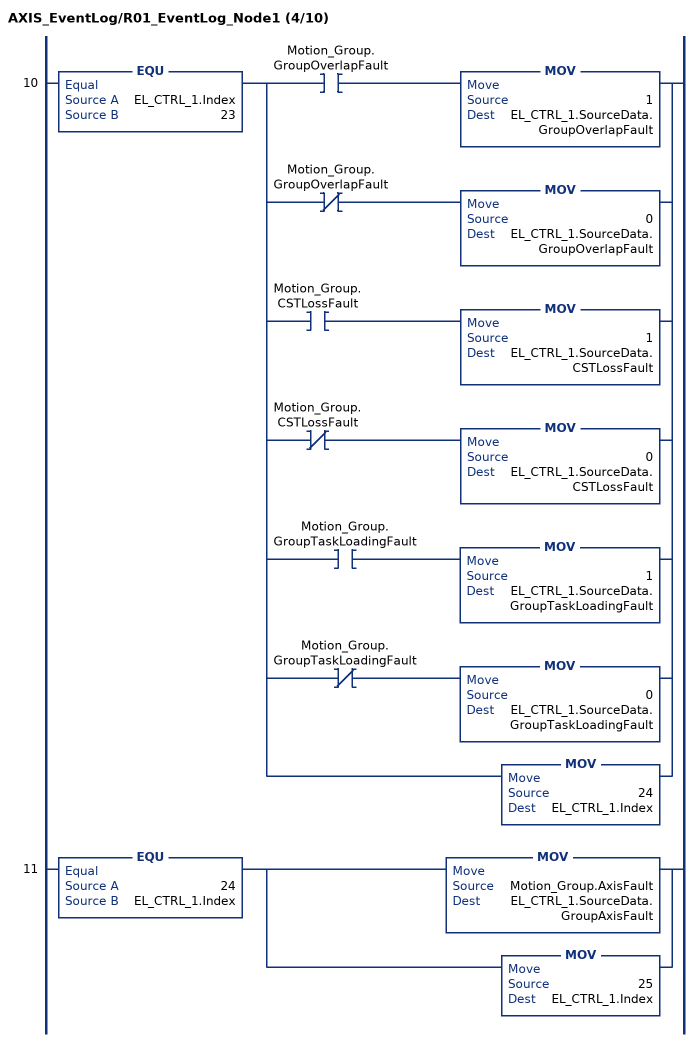
   10: EQU(EL_CTRL_1.Index,23)[XIC(Motion_Group.GroupOverlapFault) MOV(1,EL_CTRL_1.SourceData.GroupOverlapFault) ,XIO(Motion_Group.GroupOverlapFault) MOV(0,EL_CTRL_1.SourceData.GroupOverlapFault) ,XIC(Motion_Group.CSTLossFault) MOV(1,EL_CTRL_1.SourceData.CSTLossFault) ,XIO(Motion_Group.CSTLossFault) MOV(0,EL_CTRL_1.SourceData.CSTLossFault) ,XIC(Motion_Group.GroupTaskLoadingFault) MOV(1,EL_CTRL_1.SourceData.GroupTaskLoadingFault) ,XIO(Motion_Group.GroupTaskLoadingFault) MOV(0,EL_CTRL_1.SourceData.GroupTaskLoadingFault) ,MOV(24,EL_CTRL_1.Index) ];
   11: EQU(24,EL_CTRL_1.Index)[MOV(Motion_Group.AxisFault,EL_CTRL_1.SourceData.GroupAxisFault) ,MOV(25,EL_CTRL_1.Index) ];
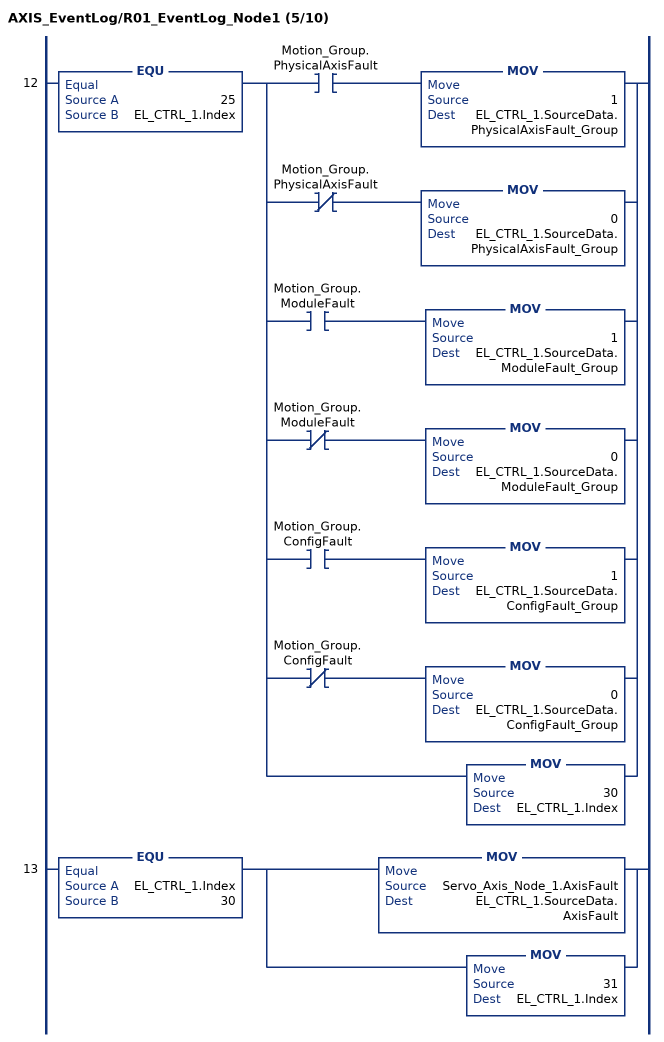
   12: EQU(25,EL_CTRL_1.Index)[XIC(Motion_Group.PhysicalAxisFault) MOV(1,EL_CTRL_1.SourceData.PhysicalAxisFault_Group) ,XIO(Motion_Group.PhysicalAxisFault) MOV(0,EL_CTRL_1.SourceData.PhysicalAxisFault_Group) ,XIC(Motion_Group.ModuleFault) MOV(1,EL_CTRL_1.SourceData.ModuleFault_Group) ,XIO(Motion_Group.ModuleFault) MOV(0,EL_CTRL_1.SourceData.ModuleFault_Group) ,XIC(Motion_Group.ConfigFault) MOV(1,EL_CTRL_1.SourceData.ConfigFault_Group) ,XIO(Motion_Group.ConfigFault) MOV(0,EL_CTRL_1.SourceData.ConfigFault_Group) ,MOV(30,EL_CTRL_1.Index) ];
   13: EQU(EL_CTRL_1.Index,30)[MOV(Servo_Axis_Node_1.AxisFault,EL_CTRL_1.SourceData.AxisFault) ,MOV(31,EL_CTRL_1.Index) ];
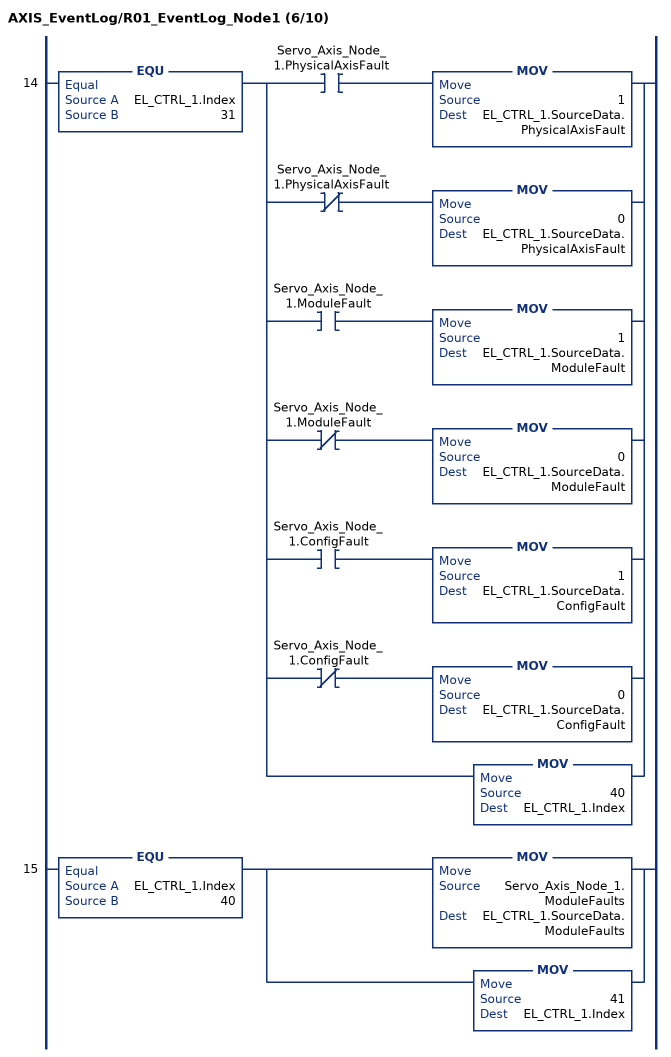
   14: EQU(EL_CTRL_1.Index,31)[XIC(Servo_Axis_Node_1.PhysicalAxisFault) MOV(1,EL_CTRL_1.SourceData.PhysicalAxisFault) ,XIO(Servo_Axis_Node_1.PhysicalAxisFault) MOV(0,EL_CTRL_1.SourceData.PhysicalAxisFault) ,XIC(Servo_Axis_Node_1.ModuleFault) MOV(1,EL_CTRL_1.SourceData.ModuleFault) ,XIO(Servo_Axis_Node_1.ModuleFault) MOV(0,EL_CTRL_1.SourceData.ModuleFault) ,XIC(Servo_Axis_Node_1.ConfigFault) MOV(1,EL_CTRL_1.SourceData.ConfigFault) ,XIO(Servo_Axis_Node_1.ConfigFault) MOV(0,EL_CTRL_1.SourceData.ConfigFault) ,MOV(40,EL_CTRL_1.Index) ];
   15: EQU(EL_CTRL_1.Index,40)[MOV(Servo_Axis_Node_1.ModuleFaults,EL_CTRL_1.SourceData.ModuleFaults) ,MOV(41,EL_CTRL_1.Index) ];
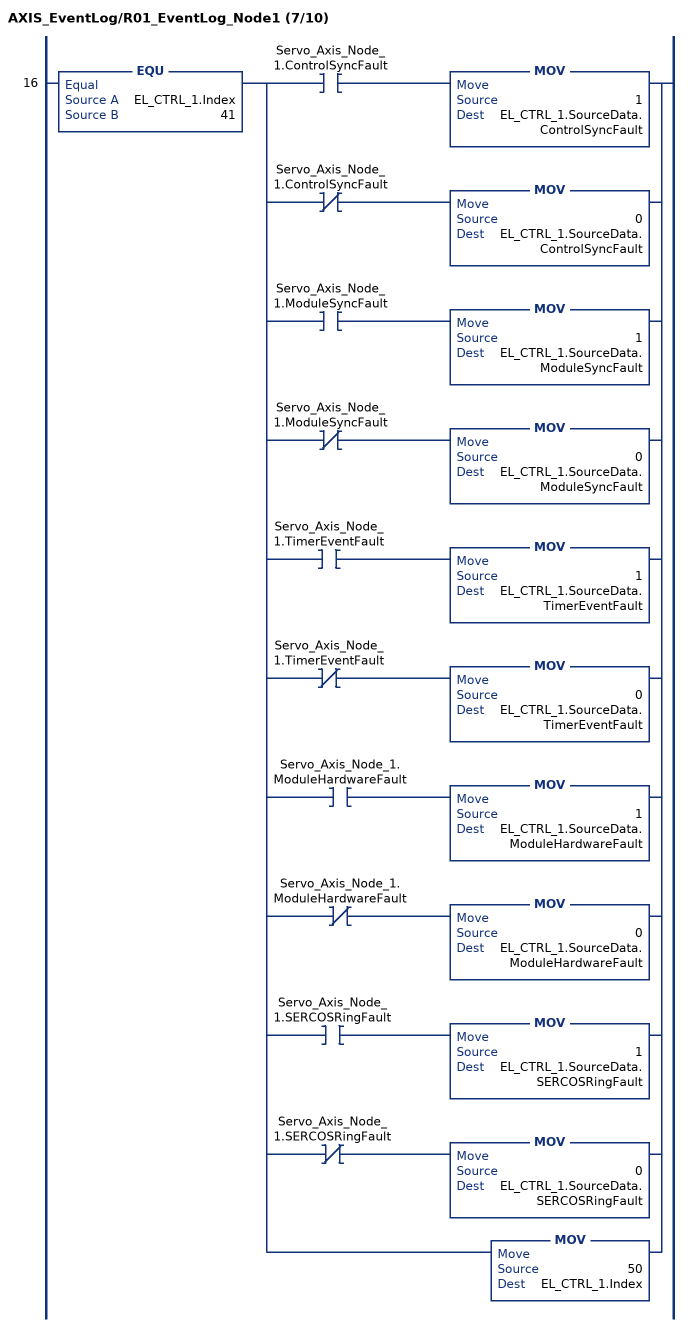
   16: EQU(EL_CTRL_1.Index,41)[XIC(Servo_Axis_Node_1.ControlSyncFault) MOV(1,EL_CTRL_1.SourceData.ControlSyncFault) ,XIO(Servo_Axis_Node_1.ControlSyncFault) MOV(0,EL_CTRL_1.SourceData.ControlSyncFault) ,XIC(Servo_Axis_Node_1.ModuleSyncFault) MOV(1,EL_CTRL_1.SourceData.ModuleSyncFault) ,XIO(Servo_Axis_Node_1.ModuleSyncFault) MOV(0,EL_CTRL_1.SourceData.ModuleSyncFault) ,XIC(Servo_Axis_Node_1.TimerEventFault) MOV(1,EL_CTRL_1.SourceData.TimerEventFault) ,XIO(Servo_Axis_Node_1.TimerEventFault) MOV(0,EL_CTRL_1.SourceData.TimerEventFault) ,XIC(Servo_Axis_Node_1.ModuleHardwareFault) MOV(1,EL_CTRL_1.SourceData.ModuleHardwareFault) ,XIO(Servo_Axis_Node_1.ModuleHardwareFault) MOV(0,EL_CTRL_1.SourceData.ModuleHardwareFault) ,XIC(Servo_Axis_Node_1.SERCOSRingFault) MOV(1,EL_CTRL_1.SourceData.SERCOSRingFault) ,XIO(Servo_Axis_Node_1.SERCOSRingFault) MOV(0,EL_CTRL_1.SourceData.SERCOSRingFault) ,MOV(50,EL_CTRL_1.Index) ];
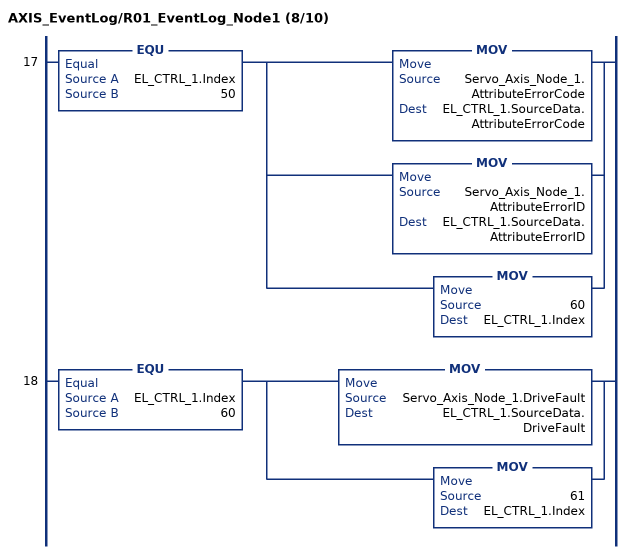
   17: EQU(EL_CTRL_1.Index,50)[MOV(Servo_Axis_Node_1.AttributeErrorCode,EL_CTRL_1.SourceData.AttributeErrorCode) ,MOV(Servo_Axis_Node_1.AttributeErrorID,EL_CTRL_1.SourceData.AttributeErrorID) ,MOV(60,EL_CTRL_1.Index) ];
   18: EQU(EL_CTRL_1.Index,60)[MOV(Servo_Axis_Node_1.DriveFault,EL_CTRL_1.SourceData.DriveFault) ,MOV(61,EL_CTRL_1.Index) ];
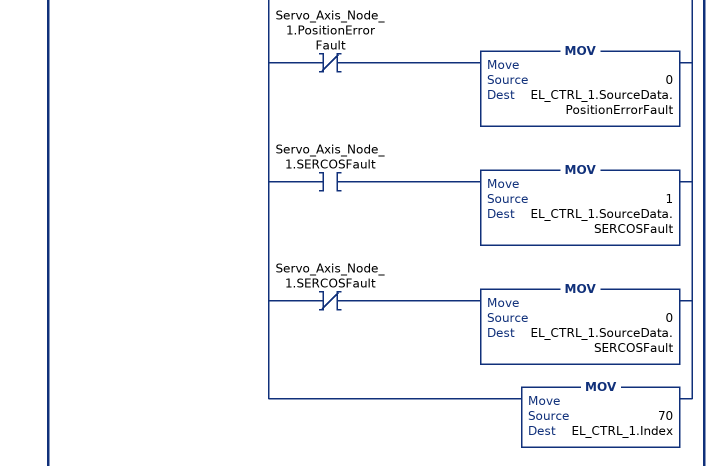
   19: EQU(EL_CTRL_1.Index,61)[XIC(Servo_Axis_Node_1.PosSoftOvertravelFault) MOV(1,EL_CTRL_1.SourceData.PosSoftOvertravelFault) ,XIO(Servo_Axis_Node_1.PosSoftOvertravelFault) MOV(0,EL_CTRL_1.SourceData.PosSoftOvertravelFault) ,XIC(Servo_Axis_Node_1.NegSoftOvertravelFault) MOV(1,EL_CTRL_1.SourceData.NegSoftOvertravelFault) ,XIO(Servo_Axis_Node_1.NegSoftOvertravelFault) MOV(0,EL_CTRL_1.SourceData.NegSoftOvertravelFault) ,XIC(Servo_Axis_Node_1.PosHardOvertravelFault) MOV(1,EL_CTRL_1.SourceData.PosHardOvertravelFault) ,XIO(Servo_Axis_Node_1.PosHardOvertravelFault) MOV(0,EL_CTRL_1.SourceData.PosHardOvertravelFault) ,XIC(Servo_Axis_Node_1.NegHardOvertravelFault) MOV(1,EL_CTRL_1.SourceData.NegHardOvertravelFault) ,XIO(Servo_Axis_Node_1.NegHardOvertravelFault) MOV(0,EL_CTRL_1.SourceData.NegHardOvertravelFault) ,XIC(Servo_Axis_Node_1.MotFeedbackFault) MOV(1,EL_CTRL_1.SourceData.MotFeedbackFault) ,XIO(Servo_Axis_Node_1.MotFeedbackFault) MOV(0,EL_CTRL_1.SourceData.MotFeedbackFault) ,XIC(Servo_Axis_Node_1.MotFeedbackNoiseFault) MOV(1,EL_CTRL_1.SourceData.MotFeedbackNoiseFault) ,XIO(Servo_Axis_Node_1.MotFeedbackNoiseFault) MOV(0,EL_CTRL_1.SourceData.MotFeedbackNoiseFault) ,XIC(Servo_Axis_Node_1.AuxFeedbackFault) MOV(1,EL_CTRL_1.SourceData.AuxFeedbackFault) ,XIO(Servo_Axis_Node_1.AuxFeedbackFault) MOV(0,EL_CTRL_1.SourceData.AuxFeedbackFault) ,XIC(Servo_Axis_Node_1.AuxFeedbackNoiseFault) MOV(1,EL_CTRL_1.SourceData.AuxFeedbackNoiseFault) ,XIO(Servo_Axis_Node_1.AuxFeedbackNoiseFault) MOV(0,EL_CTRL_1.SourceData.AuxFeedbackNoiseFault) ,XIC(Servo_Axis_Node_1.DriveEnableInputFault) MOV(1,EL_CTRL_1.SourceData.DriveEnableInputFault) ,XIO(Servo_Axis_Node_1.DriveEnableInputFault) MOV(0,EL_CTRL_1.SourceData.DriveEnableInputFault) ,XIC(Servo_Axis_Node_1.CommonBusFault) MOV(1,EL_CTRL_1.SourceData.CommonBusFault) ,XIO(Servo_Axis_Node_1.CommonBusFault) MOV(0,EL_CTRL_1.SourceData.CommonBusFault) ,XIC(Servo_Axis_Node_1.PreChargeOverloadFault) MOV(1,EL_CTRL_1.SourceData.PreChargeOverloadFault) ,XIO(Servo_Axis_Node_1.PreChargeOverloadFault) MOV(0,EL_CTRL_1.SourceData.PreChargeOverloadFault) ,XIC(Servo_Axis_Node_1.GroundShortFault) MOV(1,EL_CTRL_1.SourceData.GroundShortFault) ,XIO(Servo_Axis_Node_1.GroundShortFault) MOV(0,EL_CTRL_1.SourceData.GroundShortFault) ,XIC(Servo_Axis_Node_1.DriveHardFault) MOV(1,EL_CTRL_1.SourceData.DriveHardFault) ,XIO(Servo_Axis_Node_1.DriveHardFault) MOV(0,EL_CTRL_1.SourceData.DriveHardFault) ,XIC(Servo_Axis_Node_1.OverSpeedFault) MOV(1,EL_CTRL_1.SourceData.OverSpeedFault) ,XIO(Servo_Axis_Node_1.OverSpeedFault) MOV(0,EL_CTRL_1.SourceData.OverSpeedFault) ,XIC(Servo_Axis_Node_1.OverloadFault) MOV(1,EL_CTRL_1.SourceData.OverloadFault) ,XIO(Servo_Axis_Node_1.OverloadFault) MOV(0,EL_CTRL_1.SourceData.OverloadFault) ,XIC(Servo_Axis_Node_1.DriveOvertempFault) MOV(1,EL_CTRL_1.SourceData.DriveOvertempFault) ,XIO(Servo_Axis_Node_1.DriveOvertempFault) MOV(0,EL_CTRL_1.SourceData.DriveOvertempFault) ,XIC(Servo_Axis_Node_1.MotorOvertempFault) MOV(1,EL_CTRL_1.SourceData.MotorOvertempFault) ,XIO(Servo_Axis_Node_1.MotorOvertempFault) MOV(0,EL_CTRL_1.SourceData.MotorOvertempFault) ,XIC(Servo_Axis_Node_1.DriveCoolingFault) MOV(1,EL_CTRL_1.SourceData.DriveCoolingFault) ,XIO(Servo_Axis_Node_1.DriveCoolingFault) MOV(0,EL_CTRL_1.SourceData.DriveCoolingFault) ,XIC(Servo_Axis_Node_1.DriveControlVoltageFault) MOV(1,EL_CTRL_1.SourceData.DriveControlVoltageFault) ,XIO(Servo_Axis_Node_1.DriveControlVoltageFault) MOV(0,EL_CTRL_1.SourceData.DriveControlVoltageFault) ,XIC(Servo_Axis_Node_1.FeedbackFault) MOV(1,EL_CTRL_1.SourceData.FeedbackFault) ,XIO(Servo_Axis_Node_1.FeedbackFault) MOV(0,EL_CTRL_1.SourceData.FeedbackFault) ,XIC(Servo_Axis_Node_1.CommutationFault) MOV(1,EL_CTRL_1.SourceData.CommutationFault) ,XIO(Servo_Axis_Node_1.CommutationFault) MOV(0,EL_CTRL_1.SourceData.CommutationFault) ,XIC(Servo_Axis_Node_1.DriveOvercurrentFault) MOV(1,EL_CTRL_1.SourceData.DriveOvercurrentFault) ,XIO(Servo_Axis_Node_1.DriveOvercurrentFault) MOV(0,EL_CTRL_1.SourceData.DriveOvercurrentFault) ,XIC(Servo_Axis_Node_1.DriveOvervoltageFault) MOV(1,EL_CTRL_1.SourceData.DriveOvervoltageFault) ,XIO(Servo_Axis_Node_1.DriveOvervoltageFault) MOV(0,EL_CTRL_1.SourceData.DriveOvervoltageFault) ,XIC(Servo_Axis_Node_1.DriveUndervoltageFault) MOV(1,EL_CTRL_1.SourceData.DriveUndervoltageFault) ,XIO(Servo_Axis_Node_1.DriveUndervoltageFault) MOV(0,EL_CTRL_1.SourceData.DriveUndervoltageFault) ,XIC(Servo_Axis_Node_1.PowerPhaseLossFault) MOV(1,EL_CTRL_1.SourceData.PowerPhaseLossFault) ,XIO(Servo_Axis_Node_1.PowerPhaseLossFault) MOV(0,EL_CTRL_1.SourceData.PowerPhaseLossFault) ,XIC(Servo_Axis_Node_1.PositionErrorFault) MOV(1,EL_CTRL_1.SourceData.PositionErrorFault) ,XIO(Servo_Axis_Node_1.PositionErrorFault) MOV(0,EL_CTRL_1.SourceData.PositionErrorFault) ,XIC(Servo_Axis_Node_1.SERCOSFault) MOV(1,EL_CTRL_1.SourceData.SERCOSFault) ,XIO(Servo_Axis_Node_1.SERCOSFault) MOV(0,EL_CTRL_1.SourceData.SERCOSFault) ,MOV(70,EL_CTRL_1.Index) ];
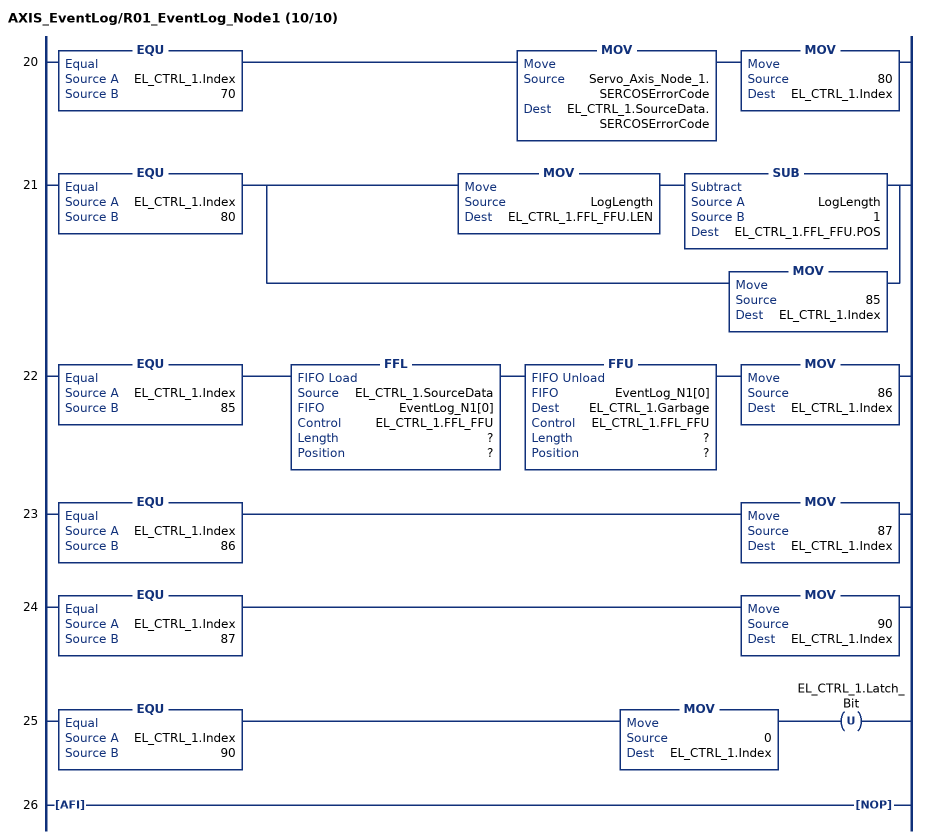
   20: EQU(EL_CTRL_1.Index,70)MOV(Servo_Axis_Node_1.SERCOSErrorCode,EL_CTRL_1.SourceData.SERCOSErrorCode)MOV(80,EL_CTRL_1.Index);
   21: EQU(EL_CTRL_1.Index,80)[MOV(LogLength,EL_CTRL_1.FFL_FFU.LEN) SUB(LogLength,1,EL_CTRL_1.FFL_FFU.POS) ,MOV(85,EL_CTRL_1.Index) ];
   22: EQU(EL_CTRL_1.Index,85)FFL(EL_CTRL_1.SourceData,EventLog_N1[0],EL_CTRL_1.FFL_FFU,?,?)FFU(EventLog_N1[0],EL_CTRL_1.Garbage,EL_CTRL_1.FFL_FFU,?,?)MOV(86,EL_CTRL_1.Index);
   23: EQU(EL_CTRL_1.Index,86)MOV(87,EL_CTRL_1.Index);
   24: EQU(EL_CTRL_1.Index,87)MOV(90,EL_CTRL_1.Index);
   25: EQU(EL_CTRL_1.Index,90)MOV(0,EL_CTRL_1.Index)OTU(EL_CTRL_1.Latch_Bit);
   26: AFI()NOP();
END_ROUTINE

ROUTINE R02_EventLog_Node2   (* ladder *)
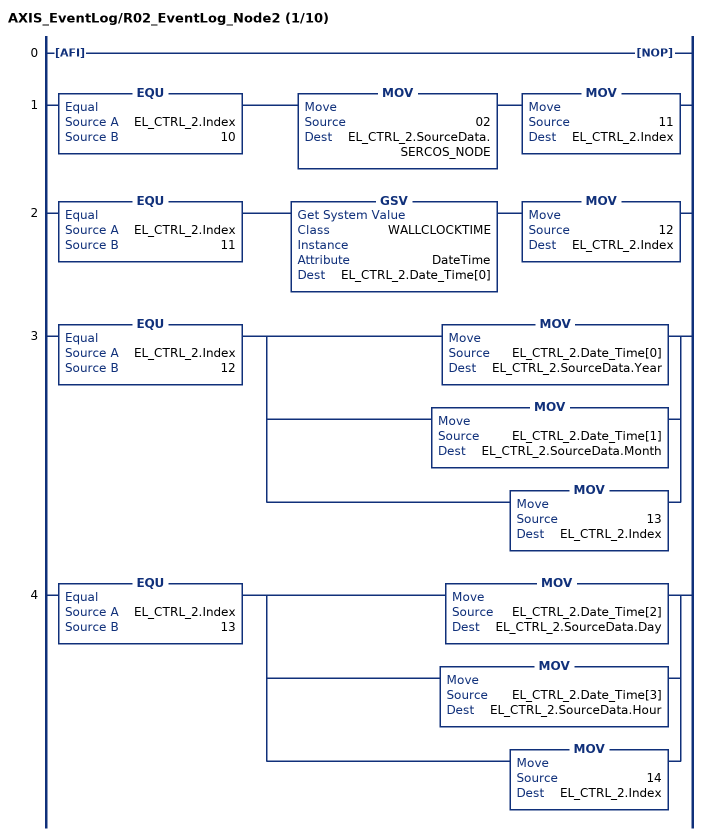
   0: AFI()NOP();
   1: EQU(EL_CTRL_2.Index,10)MOV(02,EL_CTRL_2.SourceData.SERCOS_NODE)MOV(11,EL_CTRL_2.Index);
   2: EQU(EL_CTRL_2.Index,11)GSV(WALLCLOCKTIME,,DateTime,EL_CTRL_2.Date_Time[0])MOV(12,EL_CTRL_2.Index);
   3: EQU(EL_CTRL_2.Index,12)[MOV(EL_CTRL_2.Date_Time[0],EL_CTRL_2.SourceData.Year) ,MOV(EL_CTRL_2.Date_Time[1],EL_CTRL_2.SourceData.Month) ,MOV(13,EL_CTRL_2.Index) ];
   4: EQU(EL_CTRL_2.Index,13)[MOV(EL_CTRL_2.Date_Time[2],EL_CTRL_2.SourceData.Day) ,MOV(EL_CTRL_2.Date_Time[3],EL_CTRL_2.SourceData.Hour) ,MOV(14,EL_CTRL_2.Index) ];
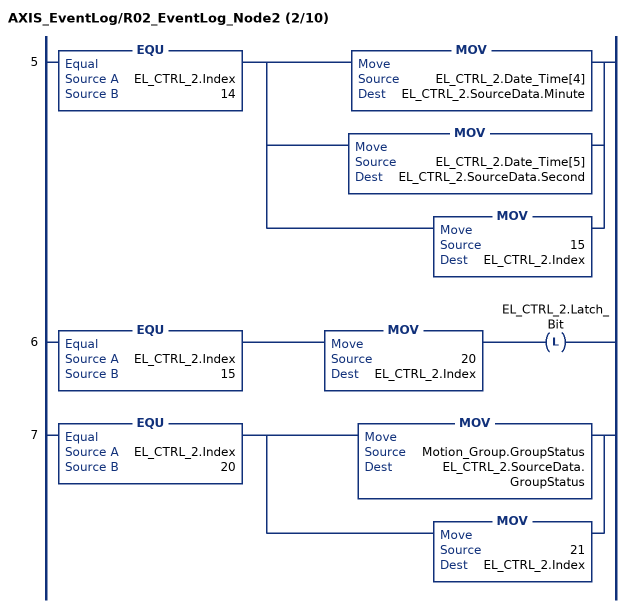
   5: EQU(EL_CTRL_2.Index,14)[MOV(EL_CTRL_2.Date_Time[4],EL_CTRL_2.SourceData.Minute) ,MOV(EL_CTRL_2.Date_Time[5],EL_CTRL_2.SourceData.Second) ,MOV(15,EL_CTRL_2.Index) ];
   6: EQU(EL_CTRL_2.Index,15)MOV(20,EL_CTRL_2.Index)OTL(EL_CTRL_2.Latch_Bit);
   7: EQU(EL_CTRL_2.Index,20)[MOV(Motion_Group.GroupStatus,EL_CTRL_2.SourceData.GroupStatus) ,MOV(21,EL_CTRL_2.Index) ];
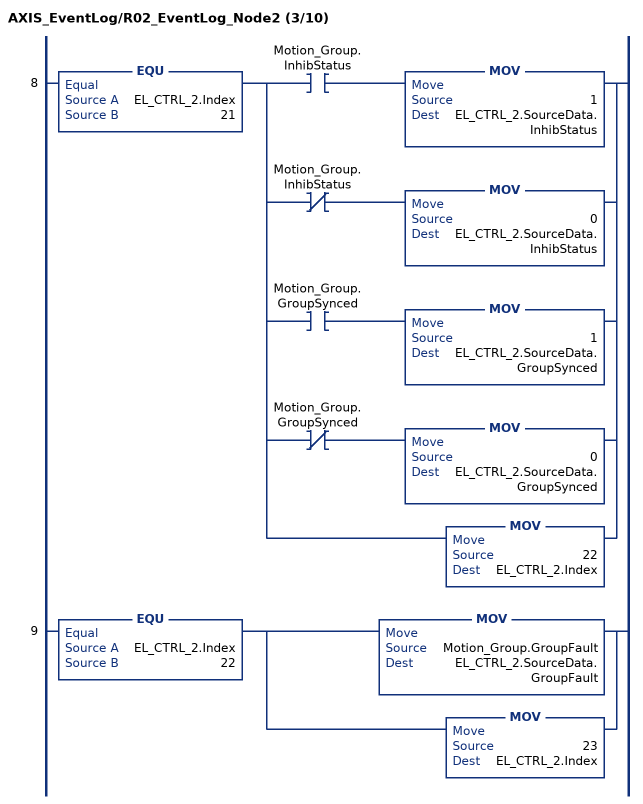
   8: EQU(EL_CTRL_2.Index,21)[XIC(Motion_Group.InhibStatus) MOV(1,EL_CTRL_2.SourceData.InhibStatus) ,XIO(Motion_Group.InhibStatus) MOV(0,EL_CTRL_2.SourceData.InhibStatus) ,XIC(Motion_Group.GroupSynced) MOV(1,EL_CTRL_2.SourceData.GroupSynced) ,XIO(Motion_Group.GroupSynced) MOV(0,EL_CTRL_2.SourceData.GroupSynced) ,MOV(22,EL_CTRL_2.Index) ];
   9: EQU(EL_CTRL_2.Index,22)[MOV(Motion_Group.GroupFault,EL_CTRL_2.SourceData.GroupFault) ,MOV(23,EL_CTRL_2.Index) ];
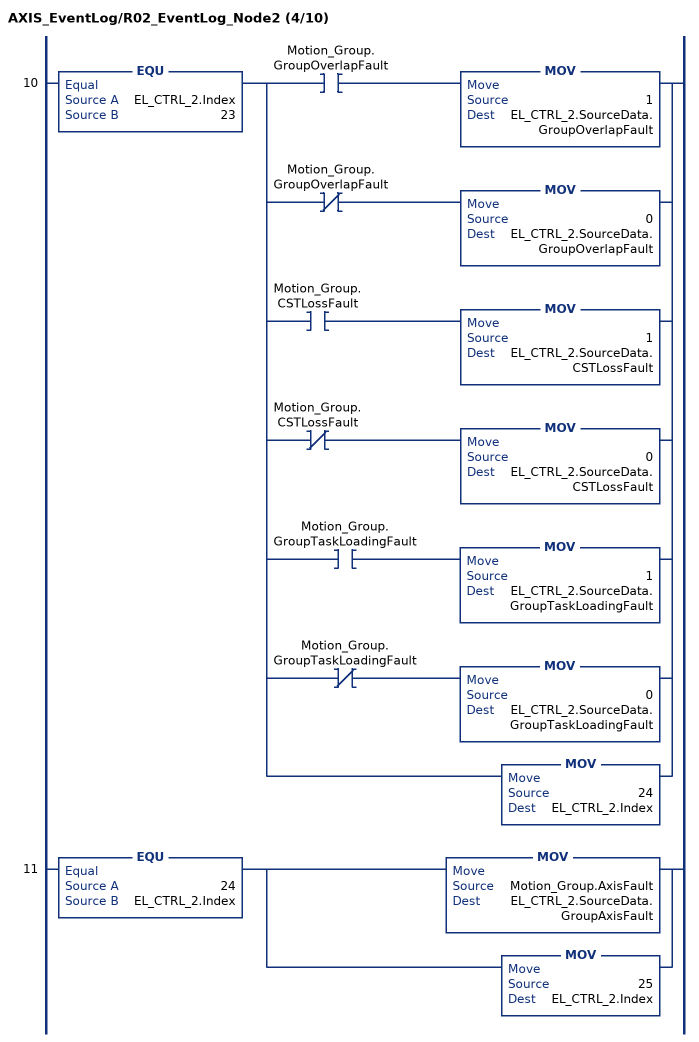
   10: EQU(EL_CTRL_2.Index,23)[XIC(Motion_Group.GroupOverlapFault) MOV(1,EL_CTRL_2.SourceData.GroupOverlapFault) ,XIO(Motion_Group.GroupOverlapFault) MOV(0,EL_CTRL_2.SourceData.GroupOverlapFault) ,XIC(Motion_Group.CSTLossFault) MOV(1,EL_CTRL_2.SourceData.CSTLossFault) ,XIO(Motion_Group.CSTLossFault) MOV(0,EL_CTRL_2.SourceData.CSTLossFault) ,XIC(Motion_Group.GroupTaskLoadingFault) MOV(1,EL_CTRL_2.SourceData.GroupTaskLoadingFault) ,XIO(Motion_Group.GroupTaskLoadingFault) MOV(0,EL_CTRL_2.SourceData.GroupTaskLoadingFault) ,MOV(24,EL_CTRL_2.Index) ];
   11: EQU(24,EL_CTRL_2.Index)[MOV(Motion_Group.AxisFault,EL_CTRL_2.SourceData.GroupAxisFault) ,MOV(25,EL_CTRL_2.Index) ];
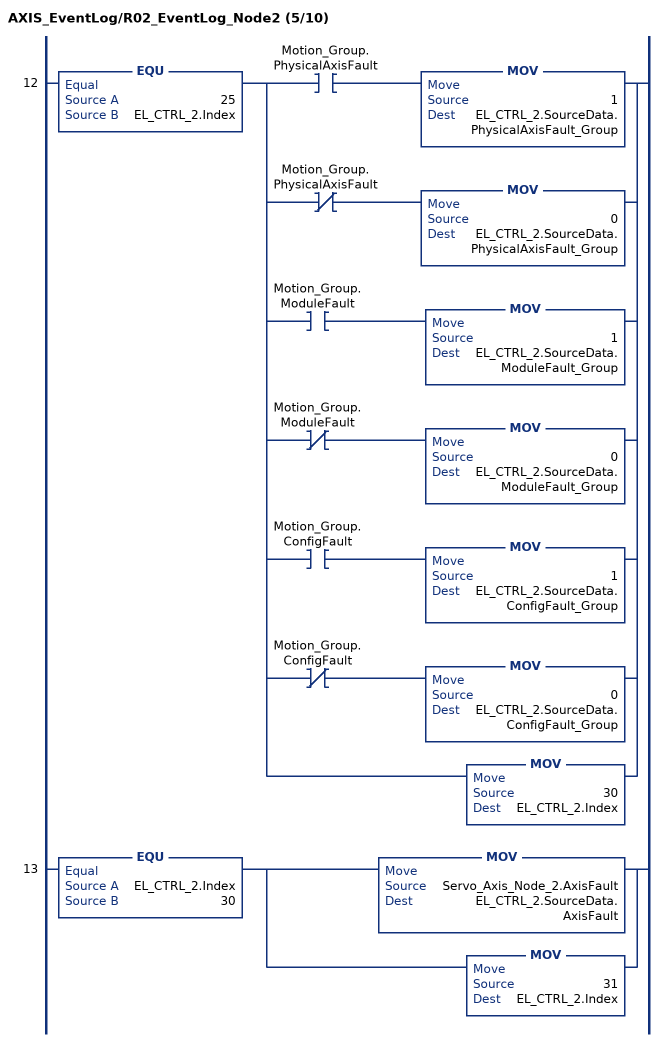
   12: EQU(25,EL_CTRL_2.Index)[XIC(Motion_Group.PhysicalAxisFault) MOV(1,EL_CTRL_2.SourceData.PhysicalAxisFault_Group) ,XIO(Motion_Group.PhysicalAxisFault) MOV(0,EL_CTRL_2.SourceData.PhysicalAxisFault_Group) ,XIC(Motion_Group.ModuleFault) MOV(1,EL_CTRL_2.SourceData.ModuleFault_Group) ,XIO(Motion_Group.ModuleFault) MOV(0,EL_CTRL_2.SourceData.ModuleFault_Group) ,XIC(Motion_Group.ConfigFault) MOV(1,EL_CTRL_2.SourceData.ConfigFault_Group) ,XIO(Motion_Group.ConfigFault) MOV(0,EL_CTRL_2.SourceData.ConfigFault_Group) ,MOV(30,EL_CTRL_2.Index) ];
   13: EQU(EL_CTRL_2.Index,30)[MOV(Servo_Axis_Node_2.AxisFault,EL_CTRL_2.SourceData.AxisFault) ,MOV(31,EL_CTRL_2.Index) ];
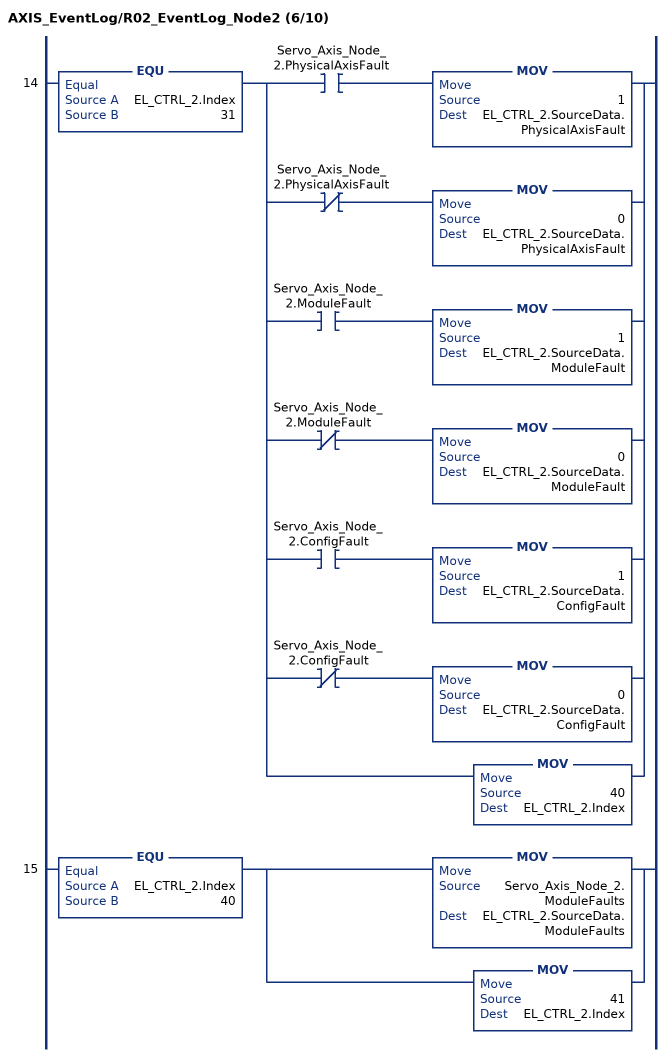
   14: EQU(EL_CTRL_2.Index,31)[XIC(Servo_Axis_Node_2.PhysicalAxisFault) MOV(1,EL_CTRL_2.SourceData.PhysicalAxisFault) ,XIO(Servo_Axis_Node_2.PhysicalAxisFault) MOV(0,EL_CTRL_2.SourceData.PhysicalAxisFault) ,XIC(Servo_Axis_Node_2.ModuleFault) MOV(1,EL_CTRL_2.SourceData.ModuleFault) ,XIO(Servo_Axis_Node_2.ModuleFault) MOV(0,EL_CTRL_2.SourceData.ModuleFault) ,XIC(Servo_Axis_Node_2.ConfigFault) MOV(1,EL_CTRL_2.SourceData.ConfigFault) ,XIO(Servo_Axis_Node_2.ConfigFault) MOV(0,EL_CTRL_2.SourceData.ConfigFault) ,MOV(40,EL_CTRL_2.Index) ];
   15: EQU(EL_CTRL_2.Index,40)[MOV(Servo_Axis_Node_2.ModuleFaults,EL_CTRL_2.SourceData.ModuleFaults) ,MOV(41,EL_CTRL_2.Index) ];
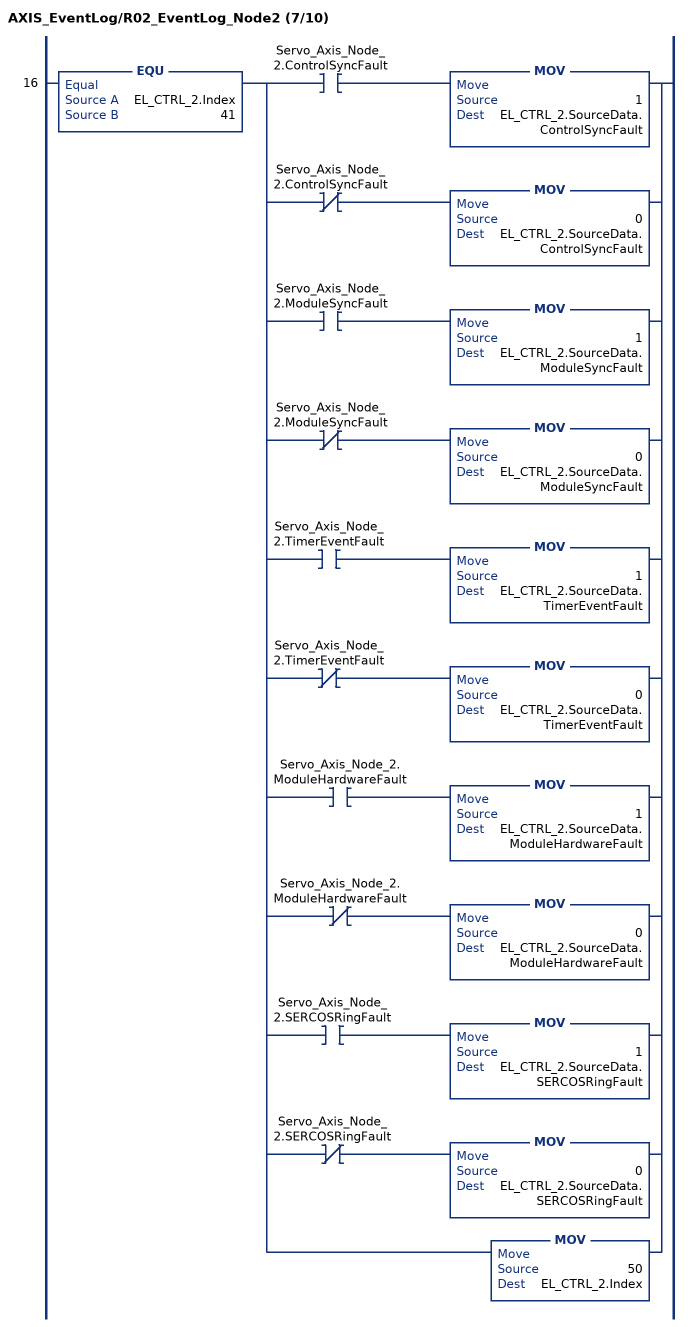
   16: EQU(EL_CTRL_2.Index,41)[XIC(Servo_Axis_Node_2.ControlSyncFault) MOV(1,EL_CTRL_2.SourceData.ControlSyncFault) ,XIO(Servo_Axis_Node_2.ControlSyncFault) MOV(0,EL_CTRL_2.SourceData.ControlSyncFault) ,XIC(Servo_Axis_Node_2.ModuleSyncFault) MOV(1,EL_CTRL_2.SourceData.ModuleSyncFault) ,XIO(Servo_Axis_Node_2.ModuleSyncFault) MOV(0,EL_CTRL_2.SourceData.ModuleSyncFault) ,XIC(Servo_Axis_Node_2.TimerEventFault) MOV(1,EL_CTRL_2.SourceData.TimerEventFault) ,XIO(Servo_Axis_Node_2.TimerEventFault) MOV(0,EL_CTRL_2.SourceData.TimerEventFault) ,XIC(Servo_Axis_Node_2.ModuleHardwareFault) MOV(1,EL_CTRL_2.SourceData.ModuleHardwareFault) ,XIO(Servo_Axis_Node_2.ModuleHardwareFault) MOV(0,EL_CTRL_2.SourceData.ModuleHardwareFault) ,XIC(Servo_Axis_Node_2.SERCOSRingFault) MOV(1,EL_CTRL_2.SourceData.SERCOSRingFault) ,XIO(Servo_Axis_Node_2.SERCOSRingFault) MOV(0,EL_CTRL_2.SourceData.SERCOSRingFault) ,MOV(50,EL_CTRL_2.Index) ];
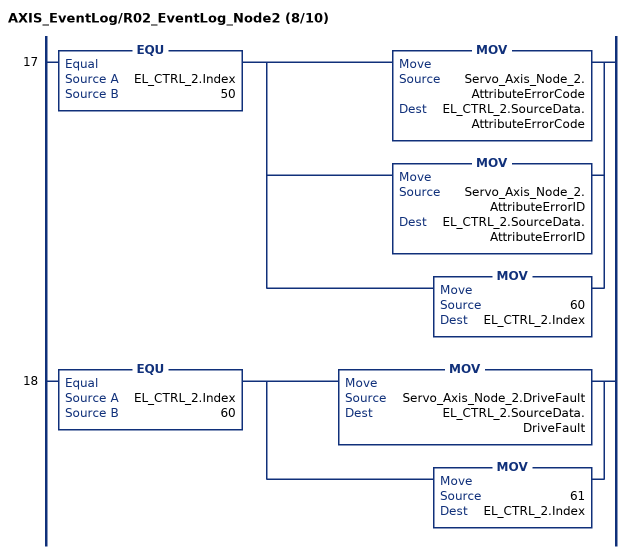
   17: EQU(EL_CTRL_2.Index,50)[MOV(Servo_Axis_Node_2.AttributeErrorCode,EL_CTRL_2.SourceData.AttributeErrorCode) ,MOV(Servo_Axis_Node_2.AttributeErrorID,EL_CTRL_2.SourceData.AttributeErrorID) ,MOV(60,EL_CTRL_2.Index) ];
   18: EQU(EL_CTRL_2.Index,60)[MOV(Servo_Axis_Node_2.DriveFault,EL_CTRL_2.SourceData.DriveFault) ,MOV(61,EL_CTRL_2.Index) ];
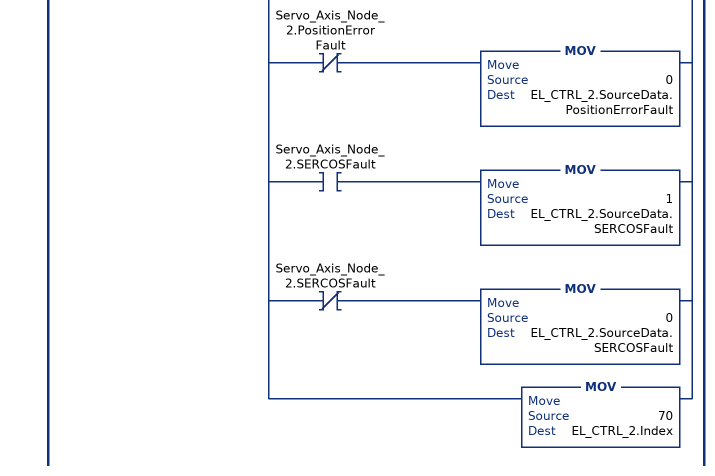
   19: EQU(EL_CTRL_2.Index,61)[XIC(Servo_Axis_Node_2.PosSoftOvertravelFault) MOV(1,EL_CTRL_2.SourceData.PosSoftOvertravelFault) ,XIO(Servo_Axis_Node_2.PosSoftOvertravelFault) MOV(0,EL_CTRL_2.SourceData.PosSoftOvertravelFault) ,XIC(Servo_Axis_Node_2.NegSoftOvertravelFault) MOV(1,EL_CTRL_2.SourceData.NegSoftOvertravelFault) ,XIO(Servo_Axis_Node_2.NegSoftOvertravelFault) MOV(0,EL_CTRL_2.SourceData.NegSoftOvertravelFault) ,XIC(Servo_Axis_Node_2.PosHardOvertravelFault) MOV(1,EL_CTRL_2.SourceData.PosHardOvertravelFault) ,XIO(Servo_Axis_Node_2.PosHardOvertravelFault) MOV(0,EL_CTRL_2.SourceData.PosHardOvertravelFault) ,XIC(Servo_Axis_Node_2.NegHardOvertravelFault) MOV(1,EL_CTRL_2.SourceData.NegHardOvertravelFault) ,XIO(Servo_Axis_Node_2.NegHardOvertravelFault) MOV(0,EL_CTRL_2.SourceData.NegHardOvertravelFault) ,XIC(Servo_Axis_Node_2.MotFeedbackFault) MOV(1,EL_CTRL_2.SourceData.MotFeedbackFault) ,XIO(Servo_Axis_Node_2.MotFeedbackFault) MOV(0,EL_CTRL_2.SourceData.MotFeedbackFault) ,XIC(Servo_Axis_Node_2.MotFeedbackNoiseFault) MOV(1,EL_CTRL_2.SourceData.MotFeedbackNoiseFault) ,XIO(Servo_Axis_Node_2.MotFeedbackNoiseFault) MOV(0,EL_CTRL_2.SourceData.MotFeedbackNoiseFault) ,XIC(Servo_Axis_Node_2.AuxFeedbackFault) MOV(1,EL_CTRL_2.SourceData.AuxFeedbackFault) ,XIO(Servo_Axis_Node_2.AuxFeedbackFault) MOV(0,EL_CTRL_2.SourceData.AuxFeedbackFault) ,XIC(Servo_Axis_Node_2.AuxFeedbackNoiseFault) MOV(1,EL_CTRL_2.SourceData.AuxFeedbackNoiseFault) ,XIO(Servo_Axis_Node_2.AuxFeedbackNoiseFault) MOV(0,EL_CTRL_2.SourceData.AuxFeedbackNoiseFault) ,XIC(Servo_Axis_Node_2.DriveEnableInputFault) MOV(1,EL_CTRL_2.SourceData.DriveEnableInputFault) ,XIO(Servo_Axis_Node_2.DriveEnableInputFault) MOV(0,EL_CTRL_2.SourceData.DriveEnableInputFault) ,XIC(Servo_Axis_Node_2.CommonBusFault) MOV(1,EL_CTRL_2.SourceData.CommonBusFault) ,XIO(Servo_Axis_Node_2.CommonBusFault) MOV(0,EL_CTRL_2.SourceData.CommonBusFault) ,XIC(Servo_Axis_Node_2.PreChargeOverloadFault) MOV(1,EL_CTRL_2.SourceData.PreChargeOverloadFault) ,XIO(Servo_Axis_Node_2.PreChargeOverloadFault) MOV(0,EL_CTRL_2.SourceData.PreChargeOverloadFault) ,XIC(Servo_Axis_Node_2.GroundShortFault) MOV(1,EL_CTRL_2.SourceData.GroundShortFault) ,XIO(Servo_Axis_Node_2.GroundShortFault) MOV(0,EL_CTRL_2.SourceData.GroundShortFault) ,XIC(Servo_Axis_Node_2.DriveHardFault) MOV(1,EL_CTRL_2.SourceData.DriveHardFault) ,XIO(Servo_Axis_Node_2.DriveHardFault) MOV(0,EL_CTRL_2.SourceData.DriveHardFault) ,XIC(Servo_Axis_Node_2.OverSpeedFault) MOV(1,EL_CTRL_2.SourceData.OverSpeedFault) ,XIO(Servo_Axis_Node_2.OverSpeedFault) MOV(0,EL_CTRL_2.SourceData.OverSpeedFault) ,XIC(Servo_Axis_Node_2.OverloadFault) MOV(1,EL_CTRL_2.SourceData.OverloadFault) ,XIO(Servo_Axis_Node_2.OverloadFault) MOV(0,EL_CTRL_2.SourceData.OverloadFault) ,XIC(Servo_Axis_Node_2.DriveOvertempFault) MOV(1,EL_CTRL_2.SourceData.DriveOvertempFault) ,XIO(Servo_Axis_Node_2.DriveOvertempFault) MOV(0,EL_CTRL_2.SourceData.DriveOvertempFault) ,XIC(Servo_Axis_Node_2.MotorOvertempFault) MOV(1,EL_CTRL_2.SourceData.MotorOvertempFault) ,XIO(Servo_Axis_Node_2.MotorOvertempFault) MOV(0,EL_CTRL_2.SourceData.MotorOvertempFault) ,XIC(Servo_Axis_Node_2.DriveCoolingFault) MOV(1,EL_CTRL_2.SourceData.DriveCoolingFault) ,XIO(Servo_Axis_Node_2.DriveCoolingFault) MOV(0,EL_CTRL_2.SourceData.DriveCoolingFault) ,XIC(Servo_Axis_Node_2.DriveControlVoltageFault) MOV(1,EL_CTRL_2.SourceData.DriveControlVoltageFault) ,XIO(Servo_Axis_Node_2.DriveControlVoltageFault) MOV(0,EL_CTRL_2.SourceData.DriveControlVoltageFault) ,XIC(Servo_Axis_Node_2.FeedbackFault) MOV(1,EL_CTRL_2.SourceData.FeedbackFault) ,XIO(Servo_Axis_Node_2.FeedbackFault) MOV(0,EL_CTRL_2.SourceData.FeedbackFault) ,XIC(Servo_Axis_Node_2.CommutationFault) MOV(1,EL_CTRL_2.SourceData.CommutationFault) ,XIO(Servo_Axis_Node_2.CommutationFault) MOV(0,EL_CTRL_2.SourceData.CommutationFault) ,XIC(Servo_Axis_Node_2.DriveOvercurrentFault) MOV(1,EL_CTRL_2.SourceData.DriveOvercurrentFault) ,XIO(Servo_Axis_Node_2.DriveOvercurrentFault) MOV(0,EL_CTRL_2.SourceData.DriveOvercurrentFault) ,XIC(Servo_Axis_Node_2.DriveOvervoltageFault) MOV(1,EL_CTRL_2.SourceData.DriveOvervoltageFault) ,XIO(Servo_Axis_Node_2.DriveOvervoltageFault) MOV(0,EL_CTRL_2.SourceData.DriveOvervoltageFault) ,XIC(Servo_Axis_Node_2.DriveUndervoltageFault) MOV(1,EL_CTRL_2.SourceData.DriveUndervoltageFault) ,XIO(Servo_Axis_Node_2.DriveUndervoltageFault) MOV(0,EL_CTRL_2.SourceData.DriveUndervoltageFault) ,XIC(Servo_Axis_Node_2.PowerPhaseLossFault) MOV(1,EL_CTRL_2.SourceData.PowerPhaseLossFault) ,XIO(Servo_Axis_Node_2.PowerPhaseLossFault) MOV(0,EL_CTRL_2.SourceData.PowerPhaseLossFault) ,XIC(Servo_Axis_Node_2.PositionErrorFault) MOV(1,EL_CTRL_2.SourceData.PositionErrorFault) ,XIO(Servo_Axis_Node_2.PositionErrorFault) MOV(0,EL_CTRL_2.SourceData.PositionErrorFault) ,XIC(Servo_Axis_Node_2.SERCOSFault) MOV(1,EL_CTRL_2.SourceData.SERCOSFault) ,XIO(Servo_Axis_Node_2.SERCOSFault) MOV(0,EL_CTRL_2.SourceData.SERCOSFault) ,MOV(70,EL_CTRL_2.Index) ];
